C05348=1007.461,339.747,-160.298,169.990,53.598,160.501
C05349=1007.467,339.963,-160.328,169.997,53.593,160.501
C05350=1007.472,340.179,-160.358,170.005,53.589,160.502
C05351=1007.477,340.395,-160.388,170.011,53.585,160.502
C05352=1007.482,340.611,-160.418,170.018,53.580,160.503
C05353=1007.489,340.859,-160.453,170.026,53.576,160.503
C05354=1007.495,341.106,-160.487,170.035,53.571,160.504
C05355=1007.501,341.354,-160.521,170.043,53.566,160.504
C05356=1007.507,341.601,-160.557,170.051,53.561,160.505
C05357=1007.513,341.849,-160.591,170.059,53.556,160.505
C05358=1007.519,342.097,-160.625,170.068,53.552,160.506
C05359=1007.526,342.344,-160.660,170.077,53.547,160.507
C05360=1007.532,342.591,-160.694,170.085,53.542,160.507
C05361=1007.537,342.840,-160.729,170.093,53.538,160.508
C05362=1007.543,343.086,-160.764,170.101,53.533,160.509
C05363=1007.550,343.334,-160.799,170.110,53.528,160.509
C05364=1007.557,343.582,-160.834,170.118,53.523,160.510
C05365=1007.562,343.829,-160.868,170.126,53.519,160.511
C05366=1007.569,344.077,-160.903,170.134,53.514,160.511
C05367=1007.575,344.325,-160.938,170.143,53.509,160.512
C05368=1007.581,344.571,-160.973,170.151,53.504,160.512
C05369=1007.588,344.819,-161.007,170.159,53.500,160.513
C05370=1007.594,345.067,-161.043,170.168,53.495,160.514
C05371=1007.600,345.314,-161.078,170.176,53.491,160.515
C05372=1007.606,345.562,-161.112,170.185,53.486,160.515
C05373=1007.612,345.809,-161.148,170.194,53.481,160.516
C05374=1007.619,346.057,-161.183,170.202,53.476,160.516
C05375=1007.625,346.304,-161.219,170.210,53.472,160.517
C05376=1007.631,346.551,-161.253,170.219,53.467,160.518
C05377=1007.637,346.799,-161.289,170.227,53.463,160.519
C05378=1007.644,347.046,-161.324,170.236,53.459,160.519
C05379=1007.651,347.294,-161.359,170.244,53.454,160.520
C05380=1007.657,347.542,-161.394,170.252,53.449,160.521
C05381=1007.663,347.789,-161.429,170.261,53.444,160.521
C05382=1007.669,348.037,-161.465,170.270,53.440,160.522
C05383=1007.676,348.283,-161.501,170.279,53.436,160.523
C05384=1007.682,348.530,-161.536,170.287,53.431,160.524
C05385=1007.366,346.389,-161.589,170.194,53.514,160.524
C05386=1007.359,346.142,-161.554,170.186,53.518,160.523
C05387=1007.353,345.894,-161.518,170.177,53.523,160.523
C05388=1007.347,345.647,-161.484,170.168,53.527,160.522
C05389=1007.341,345.399,-161.449,170.160,53.532,160.521
C05390=1007.334,345.152,-161.413,170.151,53.537,160.520
C05391=1007.328,344.905,-161.379,170.143,53.542,160.520
C05392=1007.322,344.657,-161.344,170.135,53.546,160.519
C05393=1007.316,344.410,-161.308,170.127,53.551,160.519
C05394=1007.310,344.162,-161.274,170.118,53.555,160.518
C05395=1007.303,343.915,-161.239,170.110,53.560,160.517
C05396=1007.297,343.667,-161.205,170.102,53.564,160.516
C05397=1007.291,343.420,-161.169,170.093,53.569,160.516
C05398=1007.285,343.172,-161.135,170.085,53.574,160.515
C05399=1007.279,342.925,-161.101,170.077,53.578,160.515
C05400=1007.272,342.677,-161.066,170.069,53.583,160.514
C05401=1007.266,342.429,-161.031,170.059,53.588,160.513
C05402=1007.261,342.182,-160.997,170.051,53.593,160.513
C05403=1007.254,341.934,-160.962,170.043,53.598,160.512
C05404=1007.248,341.687,-160.928,170.034,53.602,160.511
C05405=1007.241,341.439,-160.893,170.026,53.607,160.511
C05406=1007.236,341.192,-160.858,170.018,53.612,160.510
C05407=1007.230,340.944,-160.823,170.010,53.617,160.510
C05408=1007.224,340.697,-160.789,170.001,53.621,160.509
C05409=1007.218,340.450,-160.755,169.993,53.626,160.508
C05410=1007.208,340.070,-160.703,169.982,53.634,160.508
C05411=1007.199,339.691,-160.650,169.969,53.641,160.507
C05412=1007.190,339.311,-160.597,169.956,53.649,160.506
C05413=1007.180,338.932,-160.544,169.944,53.656,160.505
C05414=1007.175,338.684,-160.511,169.935,53.661,160.504
C05415=1007.169,338.437,-160.477,169.927,53.666,160.504
C05416=1007.163,338.188,-160.442,169.919,53.671,160.503
C05417=1007.157,337.941,-160.408,169.911,53.676,160.502
C05418=1007.152,337.694,-160.374,169.903,53.681,160.502
C05419=1007.145,337.446,-160.340,169.896,53.685,160.501
C05420=1007.139,337.198,-160.305,169.888,53.690,160.501
C05421=1007.134,336.951,-160.272,169.880,53.695,160.500
C05422=1007.128,336.703,-160.238,169.871,53.700,160.500
C05423=1007.122,336.456,-160.204,169.863,53.705,160.499
C05424=1007.115,336.208,-160.171,169.855,53.710,160.499
C05425=1007.109,335.960,-160.137,169.847,53.715,160.498
C05426=1007.104,335.713,-160.104,169.840,53.720,160.498
C05427=1007.098,335.465,-160.069,169.831,53.725,160.497
C05428=1007.092,335.217,-160.036,169.823,53.730,160.497
C05429=1007.086,334.969,-160.002,169.815,53.735,160.496
C05430=1007.080,334.721,-159.968,169.807,53.740,160.496
C05431=1007.074,334.474,-159.934,169.799,53.745,160.495
C05432=1007.069,334.226,-159.901,169.791,53.750,160.494
C05433=1007.062,333.979,-159.868,169.784,53.755,160.494
C05434=1007.057,333.731,-159.834,169.776,53.760,160.494
C05435=1007.051,333.484,-159.800,169.768,53.765,160.493
C05436=1007.045,333.236,-159.767,169.760,53.770,160.493
C05437=1007.040,332.988,-159.733,169.752,53.776,160.492
C05438=1007.034,332.740,-159.700,169.744,53.781,160.492
C05439=1007.028,332.493,-159.666,169.736,53.786,160.491
C05440=1007.023,332.245,-159.633,169.728,53.791,160.491
C05441=1007.017,331.997,-159.599,169.721,53.796,160.490
C05442=1007.011,331.750,-159.566,169.713,53.801,160.490
C05443=1007.005,331.502,-159.533,169.705,53.806,160.489
C05444=1006.999,331.255,-159.499,169.698,53.812,160.489
C05445=1006.994,331.007,-159.466,169.689,53.817,160.488
C05446=1006.988,330.759,-159.433,169.682,53.822,160.488
C05447=1006.982,330.511,-159.400,169.675,53.827,160.488
C05448=1006.976,330.263,-159.367,169.667,53.832,160.487
C05449=1006.972,330.016,-159.334,169.659,53.837,160.487
C05450=1006.965,329.768,-159.301,169.651,53.842,160.486
C05451=1006.960,329.520,-159.267,169.643,53.848,160.486
C05452=1006.954,329.273,-159.234,169.635,53.853,160.485
C05453=1006.948,329.025,-159.201,169.629,53.858,160.485
C05454=1006.942,328.777,-159.168,169.620,53.863,160.484
C05455=1006.937,328.530,-159.136,169.613,53.869,160.484
C05456=1006.931,328.282,-159.103,169.605,53.874,160.483
C05457=1006.926,328.034,-159.070,169.597,53.879,160.483
C05458=1006.919,327.786,-159.037,169.589,53.885,160.483
C05459=1006.915,327.538,-159.005,169.582,53.890,160.482
C05460=1006.909,327.290,-158.971,169.575,53.895,160.482
C05461=1006.903,327.043,-158.939,169.567,53.900,160.481
C05462=1006.897,326.795,-158.905,169.559,53.906,160.481
C05463=1006.893,326.547,-158.873,169.552,53.911,160.481
C05464=1006.886,326.300,-158.840,169.544,53.916,160.480
C05465=1006.881,326.051,-158.808,169.537,53.922,160.480
C05466=1006.876,325.804,-158.775,169.529,53.927,160.480
C05467=1006.870,325.556,-158.742,169.521,53.932,160.479
C05468=1006.865,325.308,-158.710,169.514,53.938,160.479
C05469=1006.859,325.061,-158.677,169.507,53.943,160.478
C05470=1006.852,324.704,-158.630,169.495,53.951,160.478
C05471=1006.844,324.349,-158.583,169.485,53.959,160.477
C05472=1006.835,323.993,-158.538,169.474,53.967,160.477
C05473=1006.827,323.638,-158.491,169.464,53.974,160.476
C05474=1006.822,323.391,-158.460,169.456,53.980,160.476
C05475=1006.816,323.142,-158.428,169.449,53.985,160.476
C05476=1006.810,322.895,-158.396,169.441,53.990,160.475
C05477=1006.805,322.646,-158.363,169.434,53.996,160.475
C05478=1006.800,322.399,-158.332,169.426,54.001,160.474
C05479=1006.794,322.151,-158.300,169.419,54.007,160.474
C05480=1006.788,321.903,-158.268,169.411,54.013,160.474
C05481=1006.782,321.655,-158.236,169.404,54.018,160.474
C05482=1006.778,321.407,-158.204,169.397,54.024,160.473
C05483=1006.772,321.159,-158.172,169.389,54.029,160.473
C05484=1006.766,320.911,-158.140,169.382,54.035,160.473
C05485=1006.760,320.663,-158.108,169.375,54.040,160.472
C05486=1006.755,320.416,-158.076,169.367,54.046,160.472
C05487=1006.749,320.168,-158.045,169.360,54.051,160.472
C05488=1006.744,319.920,-158.012,169.353,54.057,160.471
C05489=1006.739,319.672,-157.980,169.345,54.062,160.471
C05490=1006.733,319.424,-157.949,169.338,54.068,160.471
C05491=1006.727,319.176,-157.917,169.330,54.074,160.470
C05492=1006.722,318.928,-157.886,169.324,54.079,160.470
C05493=1006.717,318.681,-157.854,169.316,54.085,160.470
C05494=1006.712,318.432,-157.821,169.308,54.090,160.469
C05495=1006.706,318.185,-157.790,169.302,54.096,160.469
C05496=1006.701,317.937,-157.758,169.294,54.101,160.469
C05497=1006.696,317.689,-157.727,169.287,54.108,160.469
C05498=1006.690,317.441,-157.695,169.280,54.113,160.468
C05499=1006.685,317.193,-157.663,169.273,54.118,160.468
C05500=1006.680,316.945,-157.632,169.265,54.124,160.468
C05501=1006.675,316.697,-157.600,169.258,54.129,160.467
C05502=1006.669,316.450,-157.569,169.251,54.135,160.467
C05503=1006.664,316.202,-157.538,169.244,54.141,160.467
C05504=1006.658,315.953,-157.506,169.237,54.147,160.467
C05505=1006.654,315.705,-157.474,169.229,54.152,160.466
C05506=1006.649,315.457,-157.442,169.223,54.158,160.466
C05507=1006.643,315.209,-157.411,169.215,54.163,160.466
C05508=1006.638,314.962,-157.380,169.208,54.170,160.466
C05509=1006.633,314.714,-157.348,169.201,54.175,160.465
C05510=1006.628,314.466,-157.317,169.194,54.181,160.465
C05511=1006.623,314.218,-157.286,169.187,54.187,160.465
C05512=1006.618,313.970,-157.254,169.180,54.192,160.465
C05513=1006.613,313.722,-157.223,169.172,54.198,160.464
C05514=1006.607,313.475,-157.191,169.166,54.204,160.464
C05515=1006.602,313.226,-157.160,169.159,54.210,160.464
C05516=1006.598,312.979,-157.128,169.152,54.215,160.464
C05517=1006.593,312.730,-157.097,169.145,54.221,160.464
C05518=1006.588,312.482,-157.066,169.137,54.227,160.463
C05519=1006.582,312.235,-157.035,169.130,54.232,160.463
C05520=1006.577,311.987,-157.004,169.123,54.238,160.463
C05521=1006.572,311.739,-156.973,169.117,54.244,160.463
C05522=1006.568,311.490,-156.941,169.110,54.250,160.462
C05523=1006.562,311.243,-156.910,169.102,54.256,160.462
C05524=1006.557,310.994,-156.879,169.095,54.261,160.462
C05525=1006.553,310.747,-156.848,169.088,54.267,160.462
C05526=1006.548,310.499,-156.817,169.082,54.273,160.461
C05527=1006.543,310.251,-156.786,169.074,54.279,160.461
C05528=1006.538,310.003,-156.754,169.068,54.284,160.461
C05529=1006.533,309.755,-156.723,169.061,54.291,160.461
C05530=1006.526,309.405,-156.679,169.051,54.299,160.461
C05531=1006.519,309.055,-156.635,169.041,54.307,160.460
C05532=1006.512,308.706,-156.592,169.032,54.316,160.460
C05533=1006.505,308.356,-156.549,169.022,54.324,160.460
C05534=1006.501,308.107,-156.517,169.015,54.329,160.460
C05535=1006.496,307.860,-156.487,169.008,54.336,160.459
C05536=1006.491,307.612,-156.456,169.000,54.341,160.459
C05537=1006.485,307.364,-156.426,168.994,54.347,160.459
C05538=1006.481,307.116,-156.396,168.987,54.354,160.459
C05539=1006.475,306.868,-156.366,168.981,54.359,160.459
C05540=1006.470,306.620,-156.335,168.973,54.365,160.458
C05541=1006.465,306.373,-156.306,168.967,54.371,160.458
C05542=1006.460,306.124,-156.275,168.960,54.377,160.458
C05543=1006.454,305.876,-156.245,168.954,54.383,160.458
C05544=1006.449,305.628,-156.214,168.946,54.389,160.458
C05545=1006.444,305.380,-156.185,168.939,54.396,160.458
C05546=1006.440,305.122,-156.153,168.933,54.401,160.458
C05547=1006.434,304.865,-156.122,168.926,54.407,160.457
C05548=1006.429,304.606,-156.090,168.918,54.414,160.457
C05549=1006.423,304.348,-156.059,168.911,54.420,160.457
C05550=1006.180,304.930,-156.495,168.907,54.441,160.461
C05551=1006.187,305.298,-156.541,168.917,54.432,160.461
C05552=1006.194,305.666,-156.585,168.927,54.424,160.461
C05553=1006.203,306.035,-156.630,168.937,54.414,160.462
C05554=1006.210,306.403,-156.675,168.948,54.405,160.462
C05555=1006.215,306.650,-156.705,168.954,54.399,160.462
C05556=1006.220,306.899,-156.735,168.962,54.394,160.462
C05557=1006.225,307.147,-156.765,168.968,54.388,160.462
C05558=1006.229,307.395,-156.795,168.975,54.381,160.463
C05559=1006.235,307.643,-156.825,168.982,54.376,160.463
C05560=1006.240,307.891,-156.856,168.989,54.370,160.463
C05561=1006.245,308.138,-156.887,168.995,54.364,160.463
C05562=1006.250,308.386,-156.918,169.003,54.358,160.463
C05563=1006.257,308.739,-156.961,169.012,54.350,160.464
C05564=1006.264,309.090,-157.005,169.022,54.342,160.464
C05565=1006.270,309.442,-157.050,169.032,54.334,160.464
C05566=1006.277,309.795,-157.093,169.042,54.326,160.465
C05567=1006.282,310.043,-157.124,169.049,54.319,160.465
C05568=1006.287,310.291,-157.155,169.056,54.314,160.465
C05569=1006.293,310.539,-157.187,169.063,54.308,160.466
C05570=1006.296,310.786,-157.218,169.069,54.302,160.465
C05571=1006.301,311.035,-157.249,169.077,54.297,160.466
C05572=1006.306,311.283,-157.280,169.083,54.291,160.466
C05573=1006.312,311.531,-157.311,169.091,54.285,160.466
C05574=1006.317,311.779,-157.342,169.097,54.280,160.467
C05575=1006.321,312.027,-157.374,169.104,54.273,160.467
C05576=1006.326,312.274,-157.404,169.111,54.268,160.467
C05577=1006.331,312.522,-157.435,169.119,54.262,160.467
C05578=1006.336,312.770,-157.467,169.125,54.256,160.467
C05579=1006.341,313.018,-157.498,169.133,54.251,160.468
C05580=1006.346,313.266,-157.529,169.140,54.245,160.468
C05581=1006.351,313.514,-157.561,169.147,54.240,160.468
C05582=1006.356,313.762,-157.592,169.154,54.233,160.468
C05583=1006.361,314.010,-157.623,169.161,54.228,160.469
C05584=1006.367,314.258,-157.655,169.168,54.222,160.469
C05585=1006.372,314.506,-157.686,169.175,54.217,160.469
C05586=1006.377,314.753,-157.717,169.182,54.211,160.469
C05587=1006.381,315.002,-157.749,169.190,54.205,160.470
C05588=1006.387,315.249,-157.781,169.196,54.200,160.470
C05589=1006.392,315.497,-157.812,169.204,54.194,160.470
C05590=1006.397,315.745,-157.843,169.210,54.189,160.471
C05591=1006.402,315.993,-157.874,169.218,54.183,160.471
C05592=1006.408,316.242,-157.907,169.225,54.177,160.471
C05593=1006.413,316.490,-157.938,169.232,54.172,160.471
C05594=1006.418,316.737,-157.969,169.239,54.166,160.472
C05595=1006.423,316.985,-158.000,169.247,54.160,160.472
C05596=1006.428,317.233,-158.032,169.254,54.155,160.472
C05597=1006.434,317.480,-158.064,169.261,54.149,160.473
C05598=1006.439,317.730,-158.096,169.268,54.144,160.473
C05599=1006.444,317.977,-158.127,169.276,54.138,160.473
C05600=1006.450,318.225,-158.159,169.283,54.133,160.474
C05601=1006.455,318.473,-158.190,169.290,54.127,160.474
C05602=1006.460,318.720,-158.221,169.298,54.122,160.474
C05603=1006.466,318.968,-158.253,169.305,54.116,160.475
C05604=1006.471,319.216,-158.286,169.312,54.111,160.475
C05605=1006.476,319.464,-158.317,169.319,54.105,160.475
C05606=1006.482,319.713,-158.349,169.327,54.099,160.476
C05607=1006.487,319.960,-158.380,169.334,54.094,160.476
C05608=1006.493,320.208,-158.412,169.341,54.088,160.476
C05609=1006.498,320.456,-158.445,169.349,54.083,160.477
C05610=1006.503,320.704,-158.476,169.356,54.078,160.477
C05611=1006.509,320.951,-158.508,169.363,54.072,160.477
C05612=1006.515,321.199,-158.540,169.371,54.066,160.478
C05613=1006.520,321.447,-158.572,169.378,54.061,160.478
C05614=1006.526,321.695,-158.604,169.385,54.055,160.478
C05615=1006.531,321.943,-158.636,169.393,54.050,160.478
C05616=1006.536,322.190,-158.668,169.401,54.045,160.479
C05617=1006.542,322.439,-158.700,169.407,54.039,160.479
C05618=1006.547,322.686,-158.731,169.415,54.034,160.480
C05619=1006.553,322.934,-158.763,169.423,54.028,160.480
C05620=1006.558,323.182,-158.796,169.430,54.022,160.480
C05621=1006.564,323.430,-158.828,169.437,54.017,160.481
C05622=1006.569,323.678,-158.859,169.445,54.012,160.481
C05623=1006.578,324.036,-158.905,169.456,54.004,160.482
C05624=1006.586,324.394,-158.952,169.466,53.997,160.482
C05625=1006.594,324.752,-158.998,169.478,53.989,160.483
C05626=1006.602,325.110,-159.046,169.489,53.981,160.483
C05627=1006.607,325.358,-159.078,169.495,53.976,160.484
C05628=1006.613,325.605,-159.111,169.503,53.971,160.484
C05629=1006.618,325.854,-159.143,169.511,53.965,160.485
C05630=1006.623,326.101,-159.176,169.519,53.959,160.485
C05631=1006.629,326.348,-159.209,169.526,53.955,160.485
C05632=1006.635,326.597,-159.242,169.533,53.949,160.486
C05633=1006.639,326.844,-159.275,169.542,53.944,160.486
C05634=1006.645,327.092,-159.307,169.549,53.938,160.487
C05635=1006.651,327.340,-159.340,169.556,53.933,160.487
C05636=1006.657,327.587,-159.372,169.564,53.928,160.487
C05637=1006.662,327.836,-159.405,169.572,53.923,160.488
C05638=1006.668,328.084,-159.438,169.580,53.918,160.488
C05639=1006.674,328.331,-159.471,169.587,53.912,160.489
C05640=1006.679,328.578,-159.504,169.594,53.907,160.489
C05641=1006.684,328.827,-159.537,169.602,53.902,160.489
C05642=1006.690,329.075,-159.570,169.610,53.897,160.490
C05643=1006.696,329.322,-159.603,169.618,53.891,160.490
C05644=1006.701,329.570,-159.636,169.626,53.886,160.491
C05645=1006.707,329.817,-159.669,169.633,53.882,160.491
C05646=1006.713,330.065,-159.702,169.641,53.876,160.492
C05647=1006.719,330.313,-159.735,169.649,53.871,160.492
C05648=1006.725,330.561,-159.768,169.656,53.865,160.493
C05649=1006.730,330.809,-159.801,169.664,53.860,160.493
C05650=1006.736,331.056,-159.834,169.672,53.856,160.494
C05651=1006.741,331.303,-159.867,169.679,53.850,160.494
C05652=1006.747,331.551,-159.900,169.687,53.845,160.495
C05653=1006.752,331.799,-159.934,169.695,53.840,160.495
C05654=1006.758,332.047,-159.967,169.703,53.835,160.496
C05655=1006.764,332.295,-160.000,169.711,53.830,160.496
C05656=1006.769,332.542,-160.034,169.718,53.825,160.497
C05657=1006.775,332.790,-160.068,169.726,53.820,160.497
C05658=1006.780,333.038,-160.101,169.734,53.815,160.498
C05659=1006.787,333.286,-160.134,169.742,53.809,160.498
C05660=1006.793,333.533,-160.168,169.750,53.804,160.499
C05661=1006.798,333.781,-160.201,169.758,53.800,160.499
C05662=1006.804,334.029,-160.235,169.766,53.795,160.500
C05663=1006.810,334.276,-160.269,169.774,53.790,160.500
C05664=1006.815,334.524,-160.302,169.782,53.785,160.501
C05665=1006.821,334.771,-160.336,169.789,53.779,160.501
C05666=1006.827,335.019,-160.369,169.797,53.774,160.502
C05667=1006.833,335.268,-160.403,169.805,53.769,160.502
C05668=1006.839,335.515,-160.437,169.813,53.765,160.503
C05669=1006.845,335.763,-160.470,169.822,53.760,160.503
C05670=1006.851,336.010,-160.504,169.830,53.755,160.504
C05671=1006.857,336.257,-160.538,169.838,53.750,160.504
C05672=1006.862,336.505,-160.571,169.846,53.745,160.505
C05673=1006.869,336.753,-160.606,169.854,53.740,160.506
C05674=1006.874,337.001,-160.639,169.862,53.735,160.506
C05675=1006.880,337.248,-160.673,169.870,53.730,160.507
C05676=1006.886,337.496,-160.707,169.877,53.725,160.507
C05677=1006.892,337.744,-160.742,169.885,53.720,160.508
C05678=1006.898,337.991,-160.775,169.893,53.715,160.508
C05679=1006.904,338.239,-160.809,169.902,53.710,160.509
C05680=1006.910,338.486,-160.843,169.910,53.706,160.510
C05681=1006.916,338.734,-160.877,169.918,53.701,160.510
C05682=1006.921,338.982,-160.912,169.926,53.696,160.511
C05683=1006.929,339.306,-160.957,169.937,53.689,160.511
C05684=1006.937,339.630,-161.001,169.948,53.683,160.512
C05685=1006.945,339.955,-161.047,169.958,53.677,160.513
C05686=1006.953,340.279,-161.091,169.969,53.671,160.514
C05687=1006.959,340.527,-161.126,169.977,53.666,160.515
C05688=1006.964,340.774,-161.161,169.985,53.661,160.515
C05689=1006.971,341.022,-161.195,169.994,53.656,160.516
C05690=1006.977,341.270,-161.229,170.002,53.651,160.516
C05691=1006.983,341.518,-161.263,170.010,53.647,160.517
C05692=1006.989,341.765,-161.297,170.018,53.642,160.518
C05693=1006.995,342.013,-161.333,170.026,53.637,160.518
C05694=1007.001,342.260,-161.367,170.035,53.633,160.519
C05695=1007.007,342.508,-161.402,170.043,53.628,160.519
C05696=1007.013,342.755,-161.436,170.052,53.624,160.520
C05697=1007.020,343.003,-161.471,170.060,53.619,160.521
C05698=1007.025,343.250,-161.506,170.068,53.614,160.521
C05699=1007.032,343.498,-161.541,170.076,53.610,160.522
C05700=1007.038,343.745,-161.575,170.085,53.605,160.523
C05701=1007.044,343.993,-161.609,170.093,53.600,160.523
C05702=1007.050,344.240,-161.645,170.102,53.595,160.524
C05703=1006.736,342.085,-161.703,170.011,53.676,160.524
C05704=1006.730,341.839,-161.668,170.002,53.680,160.523
C05705=1006.724,341.591,-161.634,169.994,53.685,160.523
C05706=1006.718,341.343,-161.599,169.986,53.690,160.522
C05707=1006.713,341.096,-161.565,169.978,53.695,160.521
C05708=1006.706,340.848,-161.530,169.970,53.700,160.521
C05709=1006.700,340.600,-161.496,169.961,53.704,160.520
C05710=1006.694,340.353,-161.462,169.953,53.709,160.520
C05711=1006.688,340.105,-161.428,169.945,53.714,160.519
C05712=1006.682,339.837,-161.391,169.936,53.719,160.518
C05713=1006.676,339.568,-161.353,169.927,53.725,160.518
C05714=1006.669,339.300,-161.315,169.918,53.729,160.517
C05715=1006.663,339.031,-161.279,169.909,53.734,160.516
C05716=1006.657,338.784,-161.245,169.901,53.739,160.516
C05717=1006.651,338.536,-161.211,169.893,53.744,160.515
C05718=1006.645,338.289,-161.177,169.885,53.749,160.515
C05719=1006.639,338.041,-161.143,169.876,53.754,160.514
C05720=1006.633,337.794,-161.109,169.868,53.758,160.513
C05721=1006.628,337.545,-161.074,169.860,53.763,160.513
C05722=1006.622,337.298,-161.040,169.853,53.768,160.512
C05723=1006.616,337.050,-161.006,169.845,53.773,160.512
C05724=1006.610,336.803,-160.973,169.837,53.778,160.511
C05725=1006.604,336.556,-160.939,169.828,53.783,160.510
C05726=1006.597,336.307,-160.906,169.820,53.788,160.510
C05727=1006.592,336.060,-160.872,169.812,53.793,160.509
C05728=1006.586,335.812,-160.838,169.804,53.798,160.509
C05729=1006.580,335.565,-160.804,169.796,53.803,160.508
C05730=1006.575,335.317,-160.771,169.788,53.808,160.508
C05731=1006.569,335.069,-160.737,169.780,53.813,160.507
C05732=1006.563,334.821,-160.703,169.773,53.817,160.507
C05733=1006.557,334.574,-160.669,169.765,53.822,160.506
C05734=1006.551,334.327,-160.637,169.757,53.827,160.505
C05735=1006.546,334.079,-160.603,169.748,53.832,160.505
C05736=1006.540,333.831,-160.569,169.740,53.837,160.504
C05737=1006.534,333.583,-160.536,169.733,53.843,160.504
C05738=1006.529,333.336,-160.503,169.725,53.848,160.503
C05739=1006.523,333.088,-160.469,169.716,53.853,160.503
C05740=1006.517,332.840,-160.435,169.709,53.857,160.502
C05741=1006.512,332.592,-160.402,169.701,53.862,160.502
C05742=1006.506,332.345,-160.369,169.693,53.867,160.501
C05743=1006.500,332.097,-160.335,169.686,53.873,160.501
C05744=1006.494,331.849,-160.302,169.677,53.878,160.500
C05745=1006.489,331.601,-160.269,169.670,53.882,160.500
C05746=1006.483,331.354,-160.235,169.662,53.887,160.499
C05747=1006.477,331.106,-160.202,169.654,53.892,160.499
C05748=1006.472,330.858,-160.168,169.646,53.898,160.498
C05749=1006.467,330.611,-160.135,169.638,53.903,160.498
C05750=1006.460,330.363,-160.103,169.630,53.908,160.497
C05751=1006.455,330.115,-160.070,169.624,53.913,160.497
C05752=1006.449,329.867,-160.037,169.616,53.918,160.496
C05753=1006.443,329.619,-160.004,169.607,53.923,160.496
C05754=1006.438,329.372,-159.971,169.600,53.929,160.495
C05755=1006.432,329.124,-159.938,169.592,53.934,160.495
C05756=1006.427,328.876,-159.906,169.585,53.939,160.495
C05757=1006.421,328.628,-159.872,169.577,53.944,160.494
C05758=1006.416,328.381,-159.840,169.569,53.949,160.493
C05759=1006.410,328.133,-159.807,169.561,53.954,160.493
C05760=1006.405,327.885,-159.774,169.554,53.959,160.493
C05761=1006.399,327.638,-159.742,169.547,53.965,160.492
C05762=1006.394,327.390,-159.708,169.538,53.970,160.492
C05763=1006.388,327.142,-159.676,169.531,53.975,160.491
C05764=1006.383,326.894,-159.643,169.524,53.980,160.491
C05765=1006.377,326.646,-159.611,169.516,53.986,160.491
C05766=1006.371,326.398,-159.578,169.508,53.991,160.490
C05767=1006.366,326.151,-159.546,169.500,53.996,160.490
C05768=1006.361,325.903,-159.512,169.493,54.001,160.489
C05769=1006.355,325.656,-159.480,169.486,54.006,160.489
C05770=1006.350,325.407,-159.447,169.478,54.012,160.488
C05771=1006.345,325.159,-159.415,169.470,54.017,160.488
C05772=1006.337,324.799,-159.367,169.460,54.025,160.487
C05773=1006.329,324.439,-159.320,169.448,54.033,160.487
C05774=1006.321,324.078,-159.274,169.437,54.041,160.486
C05775=1006.312,323.719,-159.228,169.427,54.048,160.486
C05776=1006.307,323.470,-159.195,169.419,54.053,160.485
C05777=1006.302,323.222,-159.163,169.411,54.059,160.485
C05778=1006.296,322.974,-159.131,169.405,54.064,160.485
C05779=1006.290,322.727,-159.100,169.397,54.070,160.484
C05780=1006.284,322.479,-159.068,169.389,54.075,160.484
C05781=1006.280,322.231,-159.035,169.381,54.080,160.483
C05782=1006.274,321.983,-159.004,169.375,54.086,160.483
C05783=1006.268,321.735,-158.972,169.367,54.091,160.483
C05784=1006.263,321.487,-158.940,169.360,54.097,160.482
C05785=1006.257,321.239,-158.908,169.352,54.102,160.482
C05786=1006.252,320.992,-158.876,169.345,54.107,160.481
C05787=1006.247,320.744,-158.844,169.337,54.113,160.481
C05788=1006.241,320.496,-158.812,169.331,54.118,160.481
C05789=1006.235,320.248,-158.780,169.323,54.124,160.480
C05790=1006.230,320.000,-158.750,169.315,54.129,160.480
C05791=1006.224,319.752,-158.718,169.309,54.135,160.480
C05792=1006.219,319.504,-158.686,169.301,54.140,160.479
C05793=1006.214,319.257,-158.654,169.293,54.145,160.479
C05794=1006.209,319.009,-158.622,169.286,54.151,160.479
C05795=1006.203,318.760,-158.591,169.279,54.156,160.478
C05796=1006.198,318.513,-158.559,169.271,54.162,160.478
C05797=1006.193,318.265,-158.527,169.264,54.167,160.478
C05798=1006.188,318.017,-158.496,169.257,54.173,160.477
C05799=1006.183,317.769,-158.464,169.250,54.178,160.477
C05800=1006.177,317.521,-158.432,169.242,54.184,160.477
C05801=1006.172,317.273,-158.401,169.235,54.190,160.476
C05802=1006.166,317.025,-158.369,169.228,54.195,160.476
C05803=1006.161,316.777,-158.339,169.221,54.201,160.476
C05804=1006.157,316.529,-158.306,169.214,54.206,160.475
C05805=1006.152,316.281,-158.275,169.206,54.212,160.475
C05806=1006.146,316.034,-158.244,169.199,54.218,160.475
C05807=1006.141,315.786,-158.213,169.193,54.223,160.475
C05808=1006.136,315.538,-158.181,169.185,54.229,160.474
C05809=1006.131,315.290,-158.150,169.178,54.234,160.474
C05810=1006.126,315.042,-158.118,169.171,54.240,160.474
C05811=1006.121,314.794,-158.087,169.163,54.246,160.473
C05812=1006.116,314.546,-158.055,169.156,54.251,160.473
C05813=1006.110,314.298,-158.024,169.149,54.257,160.473
C05814=1006.105,314.050,-157.993,169.143,54.262,160.473
C05815=1006.101,313.802,-157.961,169.135,54.268,160.472
C05816=1006.096,313.554,-157.930,169.128,54.273,160.472
C05817=1006.091,313.306,-157.899,169.121,54.279,160.472
C05818=1006.085,313.059,-157.868,169.114,54.284,160.471
C05819=1006.080,312.810,-157.837,169.107,54.290,160.471
C05820=1006.075,312.562,-157.806,169.100,54.296,160.471
C05821=1006.071,312.314,-157.774,169.093,54.302,160.471
C05822=1006.065,312.066,-157.742,169.086,54.307,160.470
C05823=1006.061,311.819,-157.712,169.079,54.313,160.470
C05824=1006.056,311.571,-157.681,169.071,54.319,160.470
C05825=1006.051,311.323,-157.650,169.065,54.324,160.470
C05826=1006.046,311.074,-157.618,169.057,54.330,160.469
C05827=1006.041,310.826,-157.587,169.051,54.336,160.469
C05828=1006.036,310.578,-157.557,169.043,54.342,160.469
C05829=1006.031,310.331,-157.525,169.037,54.347,160.469
C05830=1006.026,310.083,-157.494,169.030,54.353,160.468
C05831=1006.021,309.835,-157.463,169.023,54.359,160.468
C05832=1006.015,309.480,-157.419,169.013,54.367,160.468
C05833=1006.008,309.126,-157.375,169.004,54.375,160.468
C05834=1006.002,308.772,-157.331,168.993,54.383,160.467
C05835=1005.994,308.417,-157.287,168.984,54.391,160.467
C05836=1005.989,308.169,-157.256,168.977,54.398,160.467
C05837=1005.985,307.922,-157.225,168.970,54.403,160.466
C05838=1005.980,307.673,-157.194,168.963,54.409,160.466
C05839=1005.975,307.426,-157.165,168.956,54.415,160.466
C05840=1005.970,307.184,-157.135,168.949,54.421,160.466
C05841=1005.965,306.942,-157.105,168.942,54.426,160.466
C05842=1005.960,306.700,-157.076,168.936,54.432,160.465
C05843=1005.955,306.459,-157.047,168.930,54.438,160.465
C05844=1005.950,306.217,-157.017,168.922,54.443,160.465
C05845=1005.945,305.976,-156.988,168.916,54.449,160.465
C05846=1005.941,305.734,-156.959,168.909,54.455,160.465
C05847=1005.935,305.492,-156.930,168.902,54.461,160.464
C05848=1005.691,306.038,-157.362,168.898,54.480,160.468
C05849=1005.698,306.392,-157.405,168.908,54.471,160.468
C05850=1005.705,306.747,-157.447,168.918,54.463,160.468
C05851=1005.713,307.102,-157.491,168.928,54.454,160.469
C05852=1005.719,307.456,-157.534,168.937,54.446,160.469
C05853=1005.725,307.704,-157.564,168.944,54.441,160.469
C05854=1005.730,307.952,-157.595,168.951,54.434,160.469
C05855=1005.735,308.200,-157.626,168.958,54.429,160.470
C05856=1005.739,308.448,-157.656,168.965,54.423,160.470
C05857=1005.746,308.805,-157.700,168.975,54.415,160.470
C05858=1005.753,309.162,-157.744,168.985,54.407,160.471
C05859=1005.760,309.517,-157.789,168.994,54.398,160.471
C05860=1005.766,309.874,-157.834,169.004,54.390,160.471
C05861=1005.772,310.122,-157.865,169.012,54.384,160.472
C05862=1005.777,310.370,-157.896,169.018,54.379,160.472
C05863=1005.781,310.619,-157.927,169.026,54.373,160.472
C05864=1005.785,310.866,-157.958,169.032,54.367,160.472
C05865=1005.790,311.114,-157.989,169.040,54.362,160.473
C05866=1005.796,311.362,-158.020,169.046,54.356,160.473
C05867=1005.801,311.611,-158.051,169.053,54.351,160.473
C05868=1005.805,311.859,-158.082,169.061,54.345,160.474
C05869=1005.809,312.106,-158.113,169.067,54.339,160.474
C05870=1005.815,312.354,-158.144,169.074,54.334,160.474
C05871=1005.820,312.602,-158.175,169.081,54.328,160.474
C05872=1005.825,312.850,-158.206,169.089,54.323,160.475
C05873=1005.830,313.098,-158.237,169.095,54.317,160.475
C05874=1005.834,313.347,-158.269,169.103,54.312,160.475
C05875=1005.839,313.594,-158.300,169.109,54.306,160.475
C05876=1005.844,313.842,-158.331,169.117,54.300,160.476
C05877=1005.849,314.090,-158.362,169.124,54.294,160.476
C05878=1005.855,314.337,-158.394,169.131,54.289,160.476
C05879=1005.860,314.586,-158.425,169.139,54.283,160.477
C05880=1005.864,314.834,-158.456,169.145,54.278,160.477
C05881=1005.870,315.081,-158.488,169.153,54.272,160.477
C05882=1005.875,315.330,-158.519,169.160,54.267,160.478
C05883=1005.880,315.578,-158.550,169.167,54.262,160.478
C05884=1005.885,315.825,-158.581,169.174,54.256,160.478
C05885=1005.889,316.074,-158.613,169.181,54.251,160.479
C05886=1005.895,316.321,-158.644,169.188,54.245,160.479
C05887=1005.900,316.569,-158.675,169.196,54.240,160.479
C05888=1005.905,316.817,-158.707,169.203,54.234,160.480
C05889=1005.911,317.066,-158.738,169.210,54.229,160.480
C05890=1005.916,317.313,-158.770,169.218,54.223,160.480
C05891=1005.921,317.562,-158.802,169.224,54.218,160.480
C05892=1005.926,317.809,-158.833,169.232,54.212,160.481
C05893=1005.931,318.057,-158.865,169.239,54.206,160.481
C05894=1005.937,318.305,-158.896,169.246,54.201,160.481
C05895=1005.942,318.552,-158.928,169.254,54.195,160.482
C05896=1005.947,318.801,-158.960,169.260,54.190,160.482
C05897=1005.952,319.049,-158.991,169.268,54.184,160.482
C05898=1005.958,319.296,-159.023,169.276,54.179,160.483
C05899=1005.963,319.544,-159.054,169.283,54.174,160.483
C05900=1005.969,319.793,-159.086,169.290,54.168,160.484
C05901=1005.974,320.040,-159.117,169.297,54.163,160.484
C05902=1005.979,320.288,-159.150,169.305,54.157,160.484
C05903=1005.984,320.536,-159.181,169.312,54.152,160.485
C05904=1005.990,320.785,-159.213,169.319,54.147,160.485
C05905=1005.995,321.032,-159.244,169.327,54.141,160.485
C05906=1006.001,321.280,-159.276,169.335,54.136,160.486
C05907=1006.006,321.528,-159.309,169.341,54.131,160.486
C05908=1006.011,321.776,-159.340,169.349,54.126,160.487
C05909=1006.017,322.023,-159.372,169.357,54.120,160.487
C05910=1006.023,322.271,-159.404,169.364,54.115,160.487
C05911=1006.028,322.519,-159.436,169.371,54.109,160.488
C05912=1006.034,322.767,-159.468,169.379,54.104,160.488
C05913=1006.039,323.015,-159.500,169.386,54.099,160.489
C05914=1006.044,323.262,-159.532,169.394,54.093,160.489
C05915=1006.050,323.511,-159.564,169.402,54.088,160.489
C05916=1006.055,323.758,-159.595,169.409,54.082,160.490
C05917=1006.064,324.121,-159.641,169.419,54.075,160.490
C05918=1006.072,324.484,-159.689,169.431,54.067,160.491
C05919=1006.080,324.846,-159.737,169.442,54.059,160.492
C05920=1006.087,325.209,-159.784,169.452,54.052,160.492
C05921=1006.093,325.457,-159.816,169.460,54.046,160.493
C05922=1006.098,325.705,-159.849,169.468,54.041,160.493
C05923=1006.104,325.953,-159.882,169.476,54.036,160.494
C05924=1006.109,326.200,-159.914,169.483,54.031,160.494
C05925=1006.114,326.448,-159.947,169.491,54.025,160.494
C05926=1006.119,326.696,-159.979,169.499,54.020,160.495
C05927=1006.125,326.943,-160.012,169.505,54.015,160.495
C05928=1006.131,327.192,-160.045,169.513,54.010,160.496
C05929=1006.136,327.439,-160.077,169.521,54.005,160.496
C05930=1006.142,327.687,-160.110,169.529,54.000,160.497
C05931=1006.147,327.935,-160.143,169.536,53.995,160.497
C05932=1006.153,328.182,-160.175,169.544,53.989,160.498
C05933=1006.158,328.431,-160.208,169.552,53.984,160.498
C05934=1006.164,328.679,-160.241,169.560,53.979,160.498
C05935=1006.169,328.925,-160.274,169.567,53.974,160.499
C05936=1006.175,329.173,-160.307,169.575,53.969,160.500
C05937=1006.180,329.422,-160.340,169.582,53.963,160.500
C05938=1006.186,329.670,-160.372,169.591,53.958,160.500
C05939=1006.191,329.917,-160.405,169.598,53.954,160.501
C05940=1006.198,330.164,-160.438,169.606,53.949,160.502
C05941=1006.203,330.412,-160.472,169.613,53.943,160.502
C05942=1006.208,330.661,-160.504,169.622,53.938,160.502
C05943=1006.214,330.908,-160.537,169.630,53.933,160.503
C05944=1006.220,331.156,-160.570,169.637,53.929,160.504
C05945=1006.225,331.403,-160.603,169.644,53.923,160.504
C05946=1006.231,331.651,-160.637,169.652,53.918,160.504
C05947=1006.237,331.899,-160.671,169.661,53.913,160.505
C05948=1006.242,332.147,-160.704,169.669,53.908,160.506
C05949=1006.248,332.394,-160.737,169.676,53.904,160.506
C05950=1006.253,332.642,-160.770,169.684,53.899,160.507
C05951=1006.258,332.890,-160.804,169.691,53.893,160.507
C05952=1006.265,333.137,-160.836,169.700,53.888,160.508
C05953=1006.270,333.385,-160.870,169.708,53.883,160.508
C05954=1006.276,333.632,-160.904,169.715,53.878,160.509
C05955=1006.282,333.880,-160.937,169.723,53.873,160.509
C05956=1006.287,334.128,-160.970,169.731,53.868,160.510
C05957=1006.293,334.375,-161.004,169.739,53.863,160.510
C05958=1006.299,334.623,-161.038,169.747,53.858,160.511
C05959=1006.304,334.871,-161.071,169.755,53.854,160.512
C05960=1006.310,335.119,-161.105,169.763,53.849,160.512
C05961=1006.316,335.366,-161.138,169.771,53.844,160.513
C05962=1006.322,335.614,-161.171,169.779,53.839,160.513
C05963=1006.328,335.862,-161.206,169.787,53.834,160.514
C05964=1006.334,336.110,-161.239,169.795,53.829,160.514
C05965=1006.340,336.357,-161.273,169.803,53.824,160.515
C05966=1006.345,336.605,-161.306,169.811,53.819,160.515
C05967=1006.351,336.852,-161.340,169.819,53.814,160.516
C05968=1006.357,337.100,-161.374,169.828,53.810,160.517
C05969=1006.362,337.348,-161.408,169.836,53.805,160.517
C05970=1006.369,337.596,-161.442,169.844,53.800,160.518
C05971=1006.375,337.843,-161.476,169.851,53.795,160.518
C05972=1006.380,338.091,-161.510,169.859,53.790,160.519
C05973=1006.386,338.338,-161.544,169.867,53.785,160.520
C05974=1006.392,338.585,-161.578,169.876,53.781,160.520
C05975=1006.398,338.834,-161.611,169.884,53.776,160.521
C05976=1006.403,339.082,-161.646,169.892,53.771,160.521
C05977=1006.409,339.293,-161.675,169.900,53.767,160.522
C05978=1006.413,339.505,-161.704,169.906,53.763,160.522
C05979=1006.419,339.717,-161.734,169.913,53.759,160.523
C05980=1006.424,339.930,-161.763,169.920,53.755,160.524
C05981=1006.113,337.770,-161.827,169.831,53.833,160.523
C05982=1006.107,337.523,-161.793,169.823,53.838,160.522
C05983=1006.102,337.275,-161.758,169.814,53.842,160.522
C05984=1006.096,337.027,-161.725,169.806,53.847,160.521
C05985=1006.090,336.779,-161.690,169.799,53.852,160.521
C05986=1006.084,336.532,-161.658,169.791,53.857,160.520
C05987=1006.078,336.284,-161.624,169.783,53.862,160.519
C05988=1006.072,336.036,-161.590,169.774,53.867,160.519
C05989=1006.067,335.789,-161.557,169.766,53.872,160.518
C05990=1006.061,335.541,-161.523,169.758,53.876,160.517
C05991=1006.056,335.293,-161.490,169.750,53.881,160.517
C05992=1006.050,335.046,-161.456,169.742,53.886,160.516
C05993=1006.044,334.798,-161.422,169.734,53.890,160.516
C05994=1006.039,334.550,-161.389,169.726,53.895,160.515
C05995=1006.032,334.303,-161.356,169.718,53.900,160.515
C05996=1006.026,334.055,-161.322,169.710,53.905,160.514
C05997=1006.021,333.808,-161.289,169.702,53.910,160.513
C05998=1006.015,333.560,-161.255,169.694,53.915,160.513
C05999=1006.010,333.312,-161.222,169.687,53.920,160.512
C06000=1006.004,333.064,-161.189,169.679,53.925,160.512
C06001=1005.998,332.817,-161.155,169.671,53.930,160.511
C06002=1005.993,332.569,-161.121,169.662,53.935,160.511
C06003=1005.987,332.321,-161.088,169.654,53.940,160.510
C06004=1005.981,332.074,-161.056,169.648,53.945,160.510
C06005=1005.976,331.826,-161.022,169.640,53.950,160.509
C06006=1005.970,331.578,-160.989,169.632,53.955,160.509
C06007=1005.965,331.330,-160.956,169.623,53.960,160.508
C06008=1005.959,331.082,-160.922,169.616,53.965,160.508
C06009=1005.954,330.834,-160.889,169.608,53.970,160.507
C06010=1005.949,330.587,-160.856,169.600,53.975,160.506
C06011=1005.942,330.339,-160.823,169.592,53.980,160.506
C06012=1005.937,330.091,-160.791,169.584,53.985,160.506
C06013=1005.932,329.844,-160.758,169.577,53.990,160.505
C06014=1005.926,329.596,-160.725,169.569,53.995,160.504
C06015=1005.920,329.348,-160.692,169.562,54.001,160.504
C06016=1005.914,329.100,-160.660,169.553,54.006,160.504
C06017=1005.909,328.853,-160.627,169.546,54.010,160.503
C06018=1005.904,328.605,-160.593,169.538,54.015,160.502
C06019=1005.898,328.357,-160.561,169.531,54.021,160.502
C06020=1005.893,328.110,-160.528,169.523,54.025,160.502
C06021=1005.887,327.862,-160.495,169.515,54.030,160.501
C06022=1005.881,327.613,-160.463,169.508,54.036,160.501
C06023=1005.877,327.366,-160.430,169.500,54.041,160.500
C06024=1005.871,327.118,-160.398,169.493,54.046,160.500
C06025=1005.866,326.871,-160.365,169.485,54.051,160.499
C06026=1005.860,326.622,-160.332,169.477,54.056,160.499
C06027=1005.854,326.375,-160.300,169.470,54.061,160.498
C06028=1005.849,326.127,-160.267,169.462,54.066,160.498
C06029=1005.844,325.879,-160.234,169.454,54.072,160.497
C06030=1005.838,325.631,-160.202,169.447,54.077,160.497
C06031=1005.833,325.383,-160.170,169.439,54.082,160.496
C06032=1005.828,325.136,-160.137,169.432,54.087,160.496
C06033=1005.822,324.887,-160.105,169.423,54.092,160.495
C06034=1005.817,324.616,-160.069,169.416,54.098,160.495
C06035=1005.811,324.343,-160.033,169.407,54.104,160.495
C06036=1005.804,324.071,-159.998,169.400,54.110,160.494
C06037=1005.798,323.799,-159.964,169.391,54.116,160.494
C06038=1005.794,323.551,-159.931,169.384,54.120,160.493
C06039=1005.788,323.303,-159.899,169.376,54.126,160.493
C06040=1005.782,323.055,-159.868,169.368,54.131,160.492
C06041=1005.776,322.807,-159.836,169.361,54.136,160.492
C06042=1005.771,322.559,-159.804,169.354,54.142,160.492
C06043=1005.766,322.312,-159.772,169.346,54.147,160.491
C06044=1005.760,322.063,-159.740,169.339,54.152,160.491
C06045=1005.755,321.816,-159.708,169.331,54.158,160.490
C06046=1005.750,321.568,-159.677,169.323,54.163,160.490
C06047=1005.744,321.319,-159.645,169.317,54.168,160.490
C06048=1005.738,321.072,-159.613,169.309,54.174,160.489
C06049=1005.734,320.824,-159.581,169.302,54.179,160.489
C06050=1005.728,320.576,-159.549,169.294,54.184,160.488
C06051=1005.723,320.328,-159.518,169.287,54.190,160.488
C06052=1005.717,320.080,-159.487,169.280,54.195,160.488
C06053=1005.712,319.833,-159.455,169.272,54.200,160.487
C06054=1005.706,319.585,-159.423,169.264,54.206,160.487
C06055=1005.702,319.336,-159.391,169.258,54.211,160.486
C06056=1005.696,319.089,-159.360,169.250,54.217,160.486
C06057=1005.691,318.841,-159.328,169.243,54.222,160.486
C06058=1005.686,318.593,-159.297,169.235,54.227,160.485
C06059=1005.680,318.345,-159.265,169.229,54.232,160.485
C06060=1005.675,318.096,-159.233,169.221,54.238,160.485
C06061=1005.670,317.849,-159.202,169.213,54.244,160.484
C06062=1005.665,317.601,-159.171,169.207,54.249,160.484
C06063=1005.660,317.353,-159.139,169.199,54.255,160.484
C06064=1005.655,317.105,-159.108,169.193,54.260,160.483
C06065=1005.649,316.858,-159.077,169.185,54.266,160.483
C06066=1005.645,316.609,-159.045,169.178,54.270,160.482
C06067=1005.639,316.362,-159.013,169.170,54.276,160.482
C06068=1005.634,316.113,-158.982,169.164,54.281,160.482
C06069=1005.629,315.866,-158.951,169.156,54.287,160.481
C06070=1005.624,315.618,-158.920,169.148,54.293,160.481
C06071=1005.620,315.369,-158.888,169.142,54.298,160.481
C06072=1005.614,315.122,-158.857,169.134,54.304,160.480
C06073=1005.609,314.874,-158.826,169.127,54.309,160.480
C06074=1005.604,314.626,-158.795,169.120,54.315,160.480
C06075=1005.599,314.378,-158.763,169.113,54.320,160.479
C06076=1005.594,314.130,-158.732,169.106,54.326,160.479
C06077=1005.589,313.881,-158.701,169.099,54.331,160.479
C06078=1005.584,313.634,-158.669,169.091,54.337,160.478
C06079=1005.579,313.387,-158.638,169.085,54.342,160.478
C06080=1005.574,313.138,-158.607,169.077,54.348,160.478
C06081=1005.569,312.890,-158.576,169.070,54.353,160.478
C06082=1005.565,312.642,-158.545,169.063,54.359,160.477
C06083=1005.560,312.394,-158.514,169.057,54.365,160.477
C06084=1005.554,312.146,-158.482,169.050,54.370,160.477
C06085=1005.550,311.899,-158.452,169.042,54.376,160.476
C06086=1005.545,311.651,-158.421,169.036,54.381,160.476
C06087=1005.540,311.402,-158.390,169.028,54.387,160.476
C06088=1005.535,311.154,-158.358,169.022,54.392,160.476
C06089=1005.531,310.907,-158.328,169.014,54.398,160.475
C06090=1005.526,310.658,-158.297,169.008,54.404,160.475
C06091=1005.521,310.410,-158.266,169.000,54.409,160.475
C06092=1005.516,310.162,-158.235,168.993,54.415,160.474
C06093=1005.512,309.914,-158.204,168.986,54.420,160.474
C06094=1005.504,309.556,-158.159,168.976,54.429,160.474
C06095=1005.498,309.197,-158.115,168.966,54.437,160.473
C06096=1005.491,308.837,-158.070,168.956,54.445,160.473
C06097=1005.484,308.479,-158.025,168.947,54.453,160.473
C06098=1005.480,308.239,-157.995,168.940,54.458,160.472
C06099=1005.475,308.000,-157.966,168.933,54.464,160.472
C06100=1005.471,307.762,-157.937,168.926,54.470,160.472
C06101=1005.465,307.522,-157.908,168.920,54.475,160.472
C06102=1005.461,307.284,-157.878,168.913,54.481,160.471
C06103=1005.456,307.045,-157.849,168.906,54.486,160.471
C06104=1005.452,306.806,-157.821,168.900,54.491,160.471
C06105=1005.447,306.567,-157.791,168.894,54.497,160.471
C06106=1005.202,307.081,-158.220,168.889,54.514,160.474
C06107=1005.209,307.438,-158.263,168.899,54.506,160.474
C06108=1005.217,307.795,-158.306,168.908,54.497,160.474
C06109=1005.223,308.152,-158.350,168.919,54.490,160.475
C06110=1005.229,308.509,-158.395,168.928,54.482,160.475
C06111=1005.236,308.870,-158.439,168.938,54.473,160.475
C06112=1005.243,309.231,-158.485,168.948,54.466,160.476
C06113=1005.250,309.593,-158.530,168.959,54.457,160.476
C06114=1005.256,309.954,-158.575,168.969,54.449,160.477
C06115=1005.261,310.203,-158.605,168.975,54.443,160.477
C06116=1005.266,310.451,-158.636,168.983,54.438,160.477
C06117=1005.271,310.698,-158.666,168.989,54.432,160.478
C06118=1005.276,310.946,-158.697,168.996,54.427,160.478
C06119=1005.280,311.195,-158.729,169.004,54.421,160.478
C06120=1005.285,311.442,-158.760,169.010,54.416,160.479
C06121=1005.290,311.690,-158.790,169.018,54.410,160.479
C06122=1005.295,311.938,-158.821,169.025,54.405,160.479
C06123=1005.300,312.186,-158.853,169.032,54.399,160.480
C06124=1005.304,312.434,-158.884,169.039,54.394,160.480
C06125=1005.309,312.682,-158.915,169.045,54.389,160.480
C06126=1005.314,312.930,-158.946,169.053,54.383,160.481
C06127=1005.319,313.178,-158.977,169.060,54.378,160.481
C06128=1005.324,313.426,-159.008,169.067,54.372,160.481
C06129=1005.329,313.674,-159.039,169.074,54.367,160.481
C06130=1005.333,313.922,-159.071,169.082,54.361,160.482
C06131=1005.338,314.170,-159.102,169.088,54.356,160.482
C06132=1005.344,314.418,-159.133,169.096,54.350,160.483
C06133=1005.349,314.666,-159.164,169.103,54.345,160.483
C06134=1005.354,314.913,-159.195,169.110,54.339,160.483
C06135=1005.358,315.162,-159.227,169.117,54.334,160.483
C06136=1005.363,315.410,-159.258,169.124,54.328,160.484
C06137=1005.369,315.658,-159.289,169.131,54.323,160.484
C06138=1005.374,315.906,-159.320,169.139,54.317,160.484
C06139=1005.379,316.154,-159.351,169.145,54.312,160.485
C06140=1005.384,316.401,-159.383,169.153,54.306,160.485
C06141=1005.389,316.650,-159.415,169.160,54.301,160.486
C06142=1005.394,316.898,-159.446,169.168,54.296,160.486
C06143=1005.399,317.145,-159.477,169.174,54.290,160.486
C06144=1005.404,317.394,-159.508,169.182,54.285,160.487
C06145=1005.410,317.641,-159.540,169.189,54.279,160.487
C06146=1005.414,317.889,-159.571,169.196,54.274,160.487
C06147=1005.419,318.137,-159.603,169.203,54.269,160.488
C06148=1005.424,318.385,-159.634,169.211,54.263,160.488
C06149=1005.430,318.633,-159.666,169.219,54.258,160.489
C06150=1005.435,318.880,-159.697,169.225,54.252,160.489
C06151=1005.441,319.129,-159.729,169.233,54.247,160.489
C06152=1005.446,319.377,-159.761,169.240,54.242,160.490
C06153=1005.451,319.625,-159.792,169.248,54.236,160.490
C06154=1005.456,319.872,-159.823,169.254,54.231,160.490
C06155=1005.461,320.120,-159.855,169.262,54.226,160.491
C06156=1005.467,320.369,-159.886,169.270,54.220,160.491
C06157=1005.472,320.617,-159.919,169.277,54.215,160.492
C06158=1005.477,320.864,-159.950,169.285,54.210,160.492
C06159=1005.482,321.112,-159.982,169.291,54.205,160.492
C06160=1005.488,321.360,-160.013,169.299,54.199,160.493
C06161=1005.494,321.608,-160.045,169.307,54.194,160.493
C06162=1005.499,321.855,-160.077,169.314,54.189,160.494
C06163=1005.504,322.103,-160.109,169.322,54.184,160.494
C06164=1005.510,322.352,-160.141,169.328,54.179,160.495
C06165=1005.515,322.600,-160.172,169.336,54.173,160.495
C06166=1005.521,322.848,-160.204,169.344,54.168,160.496
C06167=1005.526,323.095,-160.236,169.351,54.163,160.496
C06168=1005.531,323.343,-160.268,169.359,54.158,160.496
C06169=1005.537,323.591,-160.300,169.367,54.152,160.497
C06170=1005.542,323.839,-160.331,169.374,54.147,160.497
C06171=1005.547,324.070,-160.362,169.380,54.142,160.497
C06172=1005.553,324.302,-160.391,169.387,54.137,160.498
C06173=1005.558,324.534,-160.421,169.395,54.132,160.499
C06174=1005.563,324.766,-160.452,169.402,54.127,160.499
C06175=1005.567,324.996,-160.482,169.409,54.123,160.499
C06176=1005.572,325.228,-160.512,169.416,54.118,160.500
C06177=1005.577,325.459,-160.542,169.423,54.113,160.500
C06178=1005.582,325.692,-160.573,169.430,54.108,160.501
C06179=1005.588,325.939,-160.605,169.438,54.103,160.501
C06180=1005.593,326.187,-160.638,169.445,54.099,160.502
C06181=1005.598,326.435,-160.671,169.453,54.093,160.502
C06182=1005.604,326.683,-160.702,169.461,54.088,160.503
C06183=1005.609,326.931,-160.735,169.468,54.083,160.503
C06184=1005.614,327.178,-160.768,169.476,54.078,160.503
C06185=1005.620,327.427,-160.800,169.484,54.073,160.504
C06186=1005.625,327.674,-160.833,169.491,54.068,160.505
C06187=1005.630,327.922,-160.866,169.499,54.062,160.505
C06188=1005.636,328.170,-160.898,169.507,54.057,160.506
C06189=1005.641,328.417,-160.931,169.514,54.053,160.506
C06190=1005.647,328.665,-160.963,169.522,54.048,160.507
C06191=1005.653,328.913,-160.997,169.530,54.042,160.507
C06192=1005.658,329.161,-161.029,169.538,54.037,160.508
C06193=1005.664,329.409,-161.062,169.545,54.033,160.508
C06194=1005.669,329.657,-161.095,169.553,54.028,160.509
C06195=1005.674,329.904,-161.127,169.560,54.022,160.509
C06196=1005.680,330.152,-161.160,169.569,54.017,160.510
C06197=1005.686,330.400,-161.193,169.576,54.012,160.510
C06198=1005.691,330.648,-161.227,169.584,54.007,160.511
C06199=1005.697,330.895,-161.259,169.592,54.002,160.511
C06200=1005.703,331.143,-161.293,169.600,53.997,160.512
C06201=1005.708,331.391,-161.325,169.607,53.993,160.512
C06202=1005.713,331.639,-161.358,169.615,53.988,160.513
C06203=1005.719,331.887,-161.392,169.623,53.983,160.514
C06204=1005.724,332.134,-161.425,169.631,53.978,160.514
C06205=1005.730,332.381,-161.459,169.638,53.973,160.514
C06206=1005.735,332.629,-161.492,169.646,53.968,160.515
C06207=1005.741,332.877,-161.526,169.654,53.963,160.515
C06208=1005.747,333.125,-161.558,169.662,53.958,160.516
C06209=1005.753,333.373,-161.592,169.669,53.953,160.517
C06210=1005.758,333.621,-161.625,169.678,53.949,160.517
C06211=1005.763,333.868,-161.658,169.686,53.944,160.518
C06212=1005.769,334.116,-161.691,169.694,53.939,160.519
C06213=1005.775,334.363,-161.725,169.702,53.934,160.519
C06214=1005.780,334.611,-161.759,169.709,53.929,160.520
C06215=1005.786,334.859,-161.792,169.718,53.924,160.520
C06216=1005.791,335.107,-161.825,169.726,53.919,160.521
C06217=1005.798,335.354,-161.859,169.734,53.914,160.521
C06218=1005.804,335.602,-161.892,169.742,53.909,160.522
C06219=1005.495,333.430,-161.961,169.654,53.985,160.521
C06220=1005.490,333.182,-161.928,169.646,53.990,160.520
C06221=1005.484,332.934,-161.894,169.638,53.994,160.520
C06222=1005.478,332.687,-161.861,169.630,53.999,160.519
C06223=1005.472,332.439,-161.828,169.622,54.004,160.518
C06224=1005.468,332.191,-161.795,169.614,54.009,160.518
C06225=1005.462,331.944,-161.762,169.607,54.014,160.517
C06226=1005.456,331.696,-161.728,169.599,54.019,160.517
C06227=1005.451,331.448,-161.695,169.591,54.024,160.516
C06228=1005.446,331.201,-161.662,169.583,54.029,160.515
C06229=1005.440,330.953,-161.629,169.576,54.033,160.515
C06230=1005.435,330.705,-161.595,169.568,54.038,160.514
C06231=1005.429,330.457,-161.563,169.559,54.043,160.514
C06232=1005.424,330.209,-161.530,169.551,54.048,160.513
C06233=1005.418,329.961,-161.497,169.544,54.053,160.513
C06234=1005.412,329.714,-161.464,169.537,54.058,160.512
C06235=1005.407,329.466,-161.432,169.528,54.063,160.512
C06236=1005.401,329.218,-161.399,169.521,54.068,160.511
C06237=1005.396,328.970,-161.367,169.513,54.073,160.511
C06238=1005.391,328.723,-161.334,169.505,54.078,160.510
C06239=1005.385,328.475,-161.301,169.497,54.083,160.509
C06240=1005.379,328.227,-161.268,169.490,54.088,160.509
C06241=1005.374,327.979,-161.235,169.482,54.093,160.509
C06242=1005.368,327.731,-161.203,169.474,54.098,160.508
C06243=1005.363,327.484,-161.170,169.467,54.103,160.508
C06244=1005.358,327.235,-161.138,169.459,54.108,160.507
C06245=1005.353,326.989,-161.105,169.451,54.114,160.507
C06246=1005.347,326.740,-161.073,169.444,54.118,160.506
C06247=1005.342,326.493,-161.041,169.436,54.123,160.505
C06248=1005.336,326.245,-161.008,169.428,54.129,160.505
C06249=1005.332,325.997,-160.976,169.421,54.133,160.505
C06250=1005.326,325.749,-160.944,169.413,54.138,160.504
C06251=1005.321,325.501,-160.911,169.407,54.144,160.504
C06252=1005.312,325.096,-160.858,169.393,54.152,160.503
C06253=1005.303,324.690,-160.805,169.381,54.160,160.502
C06254=1005.294,324.285,-160.752,169.369,54.169,160.501
C06255=1005.286,323.879,-160.700,169.356,54.177,160.500
C06256=1005.281,323.631,-160.668,169.350,54.182,160.500
C06257=1005.275,323.383,-160.636,169.342,54.187,160.500
C06258=1005.269,323.135,-160.605,169.334,54.193,160.499
C06259=1005.265,322.888,-160.572,169.327,54.198,160.499
C06260=1005.259,322.639,-160.540,169.319,54.203,160.498
C06261=1005.253,322.392,-160.509,169.311,54.208,160.498
C06262=1005.248,322.144,-160.477,169.305,54.214,160.497
C06263=1005.243,321.896,-160.446,169.296,54.219,160.497
C06264=1005.238,321.648,-160.414,169.290,54.224,160.497
C06265=1005.232,321.400,-160.382,169.282,54.229,160.496
C06266=1005.227,321.153,-160.350,169.274,54.235,160.496
C06267=1005.221,320.904,-160.319,169.267,54.240,160.495
C06268=1005.216,320.656,-160.287,169.259,54.245,160.495
C06269=1005.210,320.409,-160.256,169.253,54.250,160.494
C06270=1005.206,320.160,-160.224,169.245,54.255,160.494
C06271=1005.201,319.913,-160.192,169.238,54.260,160.494
C06272=1005.195,319.665,-160.161,169.230,54.266,160.493
C06273=1005.190,319.416,-160.129,169.223,54.271,160.493
C06274=1005.184,319.169,-160.098,169.216,54.276,160.492
C06275=1005.180,318.920,-160.066,169.208,54.282,160.492
C06276=1005.174,318.673,-160.035,169.201,54.287,160.491
C06277=1005.169,318.425,-160.004,169.193,54.292,160.491
C06278=1005.164,318.177,-159.972,169.187,54.298,160.491
C06279=1005.159,317.929,-159.941,169.178,54.303,160.490
C06280=1005.154,317.682,-159.909,169.172,54.308,160.490
C06281=1005.149,317.433,-159.878,169.164,54.314,160.489
C06282=1005.144,317.186,-159.846,169.158,54.319,160.489
C06283=1005.139,316.938,-159.815,169.149,54.324,160.489
C06284=1005.133,316.663,-159.781,169.142,54.330,160.488
C06285=1005.127,316.389,-159.746,169.135,54.336,160.488
C06286=1005.122,316.115,-159.711,169.126,54.342,160.488
C06287=1005.116,315.841,-159.677,169.118,54.348,160.487
C06288=1005.111,315.593,-159.646,169.111,54.354,160.487
C06289=1005.106,315.345,-159.615,169.104,54.358,160.486
C06290=1005.101,315.097,-159.582,169.096,54.364,160.486
C06291=1005.096,314.849,-159.551,169.089,54.369,160.486
C06292=1005.092,314.601,-159.521,169.082,54.375,160.485
C06293=1005.087,314.353,-159.490,169.075,54.380,160.485
C06294=1005.081,314.106,-159.458,169.068,54.386,160.485
C06295=1005.077,313.857,-159.427,169.061,54.391,160.484
C06296=1005.072,313.609,-159.396,169.054,54.397,160.484
C06297=1005.067,313.361,-159.365,169.047,54.402,160.484
C06298=1005.062,313.113,-159.334,169.039,54.407,160.483
C06299=1005.057,312.865,-159.303,169.032,54.413,160.483
C06300=1005.053,312.617,-159.272,169.025,54.418,160.482
C06301=1005.048,312.369,-159.241,169.019,54.423,160.482
C06302=1005.043,312.121,-159.210,169.011,54.429,160.482
C06303=1005.038,311.873,-159.179,169.004,54.434,160.481
C06304=1005.033,311.625,-159.148,168.997,54.440,160.481
C06305=1005.028,311.377,-159.117,168.990,54.445,160.481
C06306=1005.024,311.129,-159.086,168.983,54.451,160.480
C06307=1005.019,310.881,-159.055,168.976,54.456,160.480
C06308=1005.014,310.633,-159.024,168.969,54.462,160.480
C06309=1005.010,310.386,-158.994,168.962,54.467,160.479
C06310=1005.005,310.137,-158.963,168.955,54.473,160.479
C06311=1005.001,309.890,-158.932,168.949,54.479,160.479
C06312=1004.994,309.552,-158.890,168.939,54.486,160.479
C06313=1004.988,309.214,-158.848,168.929,54.494,160.478
C06314=1004.981,308.876,-158.806,168.920,54.501,160.478
C06315=1004.975,308.539,-158.764,168.910,54.508,160.477
C06316=1004.971,308.300,-158.734,168.903,54.514,160.477
C06317=1004.966,308.060,-158.705,168.897,54.520,160.477
C06318=1004.962,307.821,-158.675,168.891,54.525,160.477
C06319=1004.957,307.581,-158.646,168.884,54.530,160.476
C06320=1004.711,308.068,-159.071,168.880,54.545,160.479
C06321=1004.716,308.319,-159.102,168.886,54.540,160.479
C06322=1004.720,308.570,-159.134,168.893,54.535,160.479
C06323=1004.727,308.936,-159.179,168.903,54.526,160.480
C06324=1004.734,309.302,-159.224,168.914,54.518,160.480
C06325=1004.741,309.668,-159.270,168.923,54.510,160.481
C06326=1004.748,310.034,-159.315,168.935,54.502,160.481
C06327=1004.753,310.282,-159.346,168.941,54.497,160.482
C06328=1004.757,310.530,-159.377,168.948,54.491,160.482
C06329=1004.762,310.778,-159.408,168.955,54.486,160.482
C06330=1004.766,311.026,-159.438,168.962,54.480,160.483
C06331=1004.771,311.274,-159.469,168.969,54.475,160.483
C06332=1004.776,311.522,-159.500,168.976,54.469,160.483
C06333=1004.780,311.770,-159.531,168.983,54.464,160.483
C06334=1004.786,312.018,-159.562,168.990,54.459,160.484
C06335=1004.791,312.266,-159.593,168.997,54.453,160.484
C06336=1004.794,312.514,-159.624,169.004,54.448,160.484
C06337=1004.799,312.762,-159.655,169.011,54.442,160.485
C06338=1004.805,313.010,-159.686,169.018,54.437,160.485
C06339=1004.810,313.258,-159.717,169.025,54.432,160.486
C06340=1004.814,313.505,-159.748,169.033,54.426,160.486
C06341=1004.819,313.754,-159.780,169.039,54.421,160.486
C06342=1004.824,314.002,-159.811,169.047,54.415,160.487
C06343=1004.829,314.250,-159.841,169.054,54.410,160.487
C06344=1004.834,314.498,-159.872,169.060,54.405,160.487
C06345=1004.839,314.746,-159.903,169.069,54.400,160.488
C06346=1004.843,314.994,-159.935,169.075,54.394,160.488
C06347=1004.848,315.241,-159.966,169.083,54.389,160.489
C06348=1004.853,315.489,-159.997,169.089,54.383,160.489
C06349=1004.858,315.738,-160.028,169.097,54.378,160.489
C06350=1004.863,315.986,-160.059,169.104,54.373,160.490
C06351=1004.869,316.233,-160.091,169.111,54.368,160.490
C06352=1004.873,316.482,-160.122,169.118,54.362,160.490
C06353=1004.878,316.730,-160.153,169.125,54.357,160.491
C06354=1004.884,316.977,-160.185,169.133,54.352,160.491
C06355=1004.889,317.225,-160.216,169.140,54.346,160.492
C06356=1004.894,317.474,-160.247,169.147,54.341,160.492
C06357=1004.898,317.721,-160.279,169.155,54.336,160.493
C06358=1004.904,317.970,-160.310,169.162,54.330,160.493
C06359=1004.909,318.217,-160.342,169.169,54.325,160.493
C06360=1004.914,318.465,-160.373,169.177,54.320,160.494
C06361=1004.919,318.713,-160.404,169.184,54.315,160.494
C06362=1004.924,318.961,-160.436,169.191,54.309,160.494
C06363=1004.929,319.209,-160.467,169.198,54.305,160.495
C06364=1004.934,319.457,-160.498,169.206,54.299,160.495
C06365=1004.940,319.704,-160.530,169.213,54.294,160.496
C06366=1004.945,319.952,-160.561,169.221,54.289,160.496
C06367=1004.951,320.201,-160.593,169.228,54.284,160.497
C06368=1004.955,320.449,-160.625,169.235,54.278,160.497
C06369=1004.960,320.697,-160.656,169.242,54.273,160.497
C06370=1004.966,320.944,-160.688,169.250,54.268,160.498
C06371=1004.971,321.192,-160.719,169.258,54.262,160.498
C06372=1004.977,321.440,-160.751,169.265,54.258,160.499
C06373=1004.981,321.688,-160.783,169.273,54.252,160.499
C06374=1004.987,321.936,-160.815,169.280,54.247,160.500
C06375=1004.992,322.184,-160.846,169.287,54.242,160.500
C06376=1004.998,322.432,-160.878,169.294,54.237,160.501
C06377=1005.003,322.680,-160.909,169.302,54.231,160.501
C06378=1005.009,322.927,-160.941,169.310,54.226,160.502
C06379=1005.013,323.176,-160.973,169.317,54.222,160.502
C06380=1005.019,323.424,-161.005,169.325,54.216,160.503
C06381=1005.024,323.671,-161.036,169.332,54.211,160.503
C06382=1005.030,323.920,-161.068,169.340,54.206,160.503
C06383=1005.037,324.267,-161.113,169.350,54.199,160.504
C06384=1005.045,324.615,-161.158,169.361,54.192,160.505
C06385=1005.052,324.963,-161.204,169.372,54.185,160.506
C06386=1005.060,325.311,-161.249,169.382,54.177,160.506
C06387=1005.065,325.558,-161.282,169.390,54.172,160.507
C06388=1005.071,325.806,-161.314,169.397,54.168,160.507
C06389=1005.075,326.054,-161.346,169.405,54.162,160.508
C06390=1005.080,326.303,-161.379,169.413,54.157,160.508
C06391=1005.086,326.550,-161.411,169.420,54.152,160.509
C06392=1005.091,326.797,-161.443,169.428,54.147,160.509
C06393=1005.096,327.045,-161.477,169.436,54.142,160.510
C06394=1005.102,327.293,-161.508,169.443,54.137,160.510
C06395=1005.107,327.541,-161.541,169.451,54.132,160.511
C06396=1005.113,327.789,-161.574,169.459,54.127,160.511
C06397=1005.118,328.037,-161.606,169.466,54.123,160.512
C06398=1005.123,328.285,-161.639,169.474,54.118,160.513
C06399=1005.129,328.532,-161.671,169.481,54.113,160.513
C06400=1005.134,328.780,-161.704,169.489,54.107,160.513
C06401=1005.139,329.028,-161.736,169.497,54.102,160.514
C06402=1005.145,329.276,-161.769,169.505,54.097,160.515
C06403=1005.151,329.524,-161.802,169.512,54.093,160.515
C06404=1005.156,329.771,-161.835,169.520,54.088,160.516
C06405=1005.162,330.019,-161.867,169.528,54.083,160.516
C06406=1005.167,330.267,-161.900,169.536,54.078,160.517
C06407=1005.172,330.515,-161.933,169.544,54.073,160.517
C06408=1005.178,330.762,-161.966,169.552,54.068,160.518
C06409=1005.184,331.010,-161.999,169.559,54.064,160.519
C06410=1005.189,331.258,-162.031,169.567,54.059,160.519
C06411=1004.884,329.077,-162.106,169.480,54.131,160.517
C06412=1004.877,328.829,-162.073,169.473,54.136,160.517
C06413=1004.873,328.581,-162.041,169.465,54.141,160.516
C06414=1004.867,328.333,-162.007,169.457,54.146,160.516
C06415=1004.862,328.086,-161.976,169.450,54.151,160.515
C06416=1004.856,327.838,-161.942,169.442,54.156,160.515
C06417=1004.851,327.590,-161.910,169.435,54.160,160.514
C06418=1004.845,327.342,-161.878,169.427,54.165,160.513
C06419=1004.840,327.095,-161.845,169.419,54.170,160.513
C06420=1004.835,326.846,-161.813,169.412,54.175,160.512
C06421=1004.830,326.599,-161.781,169.404,54.180,160.512
C06422=1004.824,326.351,-161.748,169.396,54.186,160.511
C06423=1004.820,326.103,-161.715,169.389,54.190,160.511
C06424=1004.814,325.855,-161.684,169.381,54.195,160.510
C06425=1004.809,325.607,-161.650,169.374,54.200,160.510
C06426=1004.803,325.360,-161.619,169.366,54.205,160.509
C06427=1004.799,325.112,-161.586,169.359,54.210,160.509
C06428=1004.792,324.824,-161.548,169.350,54.216,160.508
C06429=1004.787,324.536,-161.511,169.341,54.222,160.508
C06430=1004.780,324.247,-161.473,169.333,54.228,160.507
C06431=1004.774,323.959,-161.437,169.323,54.233,160.506
C06432=1004.769,323.712,-161.405,169.316,54.239,160.506
C06433=1004.763,323.463,-161.373,169.309,54.244,160.505
C06434=1004.758,323.216,-161.341,169.300,54.249,160.505
C06435=1004.753,322.968,-161.309,169.293,54.254,160.504
C06436=1004.747,322.719,-161.278,169.286,54.259,160.504
C06437=1004.742,322.472,-161.246,169.278,54.264,160.503
C06438=1004.737,322.224,-161.215,169.271,54.269,160.503
C06439=1004.731,321.977,-161.183,169.263,54.274,160.502
C06440=1004.725,321.728,-161.152,169.256,54.280,160.502
C06441=1004.721,321.480,-161.119,169.248,54.285,160.501
C06442=1004.715,321.233,-161.088,169.241,54.289,160.501
C06443=1004.710,320.984,-161.057,169.233,54.295,160.501
C06444=1004.705,320.737,-161.025,169.226,54.299,160.500
C06445=1004.700,320.489,-160.994,169.219,54.305,160.500
C06446=1004.695,320.240,-160.962,169.212,54.310,160.499
C06447=1004.690,319.992,-160.931,169.204,54.315,160.499
C06448=1004.684,319.745,-160.899,169.197,54.320,160.498
C06449=1004.679,319.497,-160.867,169.189,54.326,160.498
C06450=1004.674,319.249,-160.836,169.182,54.330,160.497
C06451=1004.669,319.001,-160.805,169.174,54.336,160.497
C06452=1004.664,318.753,-160.773,169.168,54.341,160.497
C06453=1004.659,318.505,-160.742,169.160,54.346,160.496
C06454=1004.654,318.257,-160.711,169.153,54.352,160.496
C06455=1004.648,318.009,-160.680,169.145,54.357,160.495
C06456=1004.643,317.762,-160.648,169.138,54.362,160.495
C06457=1004.639,317.513,-160.616,169.130,54.367,160.494
C06458=1004.634,317.265,-160.585,169.124,54.372,160.494
C06459=1004.628,317.018,-160.554,169.116,54.378,160.494
C06460=1004.623,316.770,-160.523,169.109,54.383,160.493
C06461=1004.618,316.521,-160.492,169.101,54.388,160.493
C06462=1004.614,316.273,-160.460,169.095,54.394,160.492
C06463=1004.608,316.025,-160.429,169.087,54.398,160.492
C06464=1004.603,315.777,-160.398,169.080,54.404,160.491
C06465=1004.599,315.530,-160.367,169.073,54.409,160.491
C06466=1004.594,315.282,-160.336,169.065,54.414,160.491
C06467=1004.589,315.034,-160.304,169.058,54.420,160.490
C06468=1004.584,314.786,-160.273,169.052,54.425,160.490
C06469=1004.579,314.538,-160.242,169.044,54.431,160.490
C06470=1004.574,314.290,-160.211,169.037,54.435,160.489
C06471=1004.569,314.042,-160.181,169.029,54.441,160.489
C06472=1004.564,313.794,-160.150,169.023,54.446,160.488
C06473=1004.560,313.546,-160.118,169.016,54.452,160.488
C06474=1004.555,313.297,-160.087,169.008,54.457,160.488
C06475=1004.550,313.050,-160.057,169.001,54.462,160.487
C06476=1004.545,312.802,-160.026,168.995,54.467,160.487
C06477=1004.540,312.554,-159.995,168.987,54.473,160.487
C06478=1004.536,312.306,-159.963,168.980,54.478,160.486
C06479=1004.531,312.058,-159.933,168.973,54.484,160.486
C06480=1004.526,311.810,-159.902,168.966,54.489,160.485
C06481=1004.522,311.562,-159.871,168.959,54.494,160.485
C06482=1004.517,311.314,-159.840,168.951,54.500,160.485
C06483=1004.512,311.066,-159.808,168.945,54.505,160.484
C06484=1004.508,310.818,-159.778,168.938,54.510,160.484
C06485=1004.503,310.570,-159.748,168.931,54.516,160.484
C06486=1004.499,310.322,-159.717,168.924,54.521,160.483
C06487=1004.494,310.074,-159.686,168.917,54.527,160.483
C06488=1004.487,309.706,-159.640,168.906,54.535,160.482
C06489=1004.480,309.337,-159.595,168.896,54.543,160.482
C06490=1004.474,308.969,-159.549,168.886,54.551,160.481
C06491=1004.466,308.572,-159.500,168.876,54.559,160.481
C06492=1004.220,309.003,-159.920,168.869,54.574,160.483
C06493=1004.225,309.281,-159.953,168.877,54.568,160.483
C06494=1004.229,309.558,-159.988,168.884,54.562,160.484
C06495=1004.235,309.836,-160.022,168.893,54.556,160.484
C06496=1004.240,310.113,-160.056,168.901,54.550,160.485
C06497=1004.245,310.362,-160.088,168.907,54.545,160.485
C06498=1004.249,310.610,-160.118,168.915,54.539,160.485
C06499=1004.254,310.858,-160.149,168.921,54.534,160.486
C06500=1004.258,311.106,-160.179,168.928,54.529,160.486
C06501=1004.263,311.354,-160.210,168.935,54.523,160.486
C06502=1004.268,311.602,-160.242,168.943,54.518,160.487
C06503=1004.272,311.850,-160.272,168.949,54.513,160.487
C06504=1004.277,312.098,-160.303,168.956,54.508,160.487
C06505=1004.281,312.346,-160.333,168.964,54.502,160.488
C06506=1004.286,312.594,-160.364,168.971,54.497,160.488
C06507=1004.291,312.842,-160.396,168.977,54.492,160.489
C06508=1004.296,313.090,-160.427,168.985,54.486,160.489
C06509=1004.300,313.338,-160.457,168.992,54.481,160.489
C06510=1004.305,313.586,-160.488,168.999,54.476,160.490
C06511=1004.311,313.834,-160.519,169.007,54.471,160.490
C06512=1004.315,314.082,-160.550,169.013,54.465,160.491
C06513=1004.319,314.330,-160.581,169.020,54.460,160.491
C06514=1004.324,314.578,-160.612,169.028,54.455,160.492
C06515=1004.330,314.826,-160.644,169.035,54.450,160.492
C06516=1004.335,315.074,-160.675,169.042,54.444,160.492
C06517=1004.339,315.321,-160.705,169.049,54.439,160.493
C06518=1004.344,315.570,-160.737,169.056,54.434,160.493
C06519=1004.349,315.818,-160.768,169.064,54.428,160.493
C06520=1004.354,316.066,-160.799,169.071,54.424,160.494
C06521=1004.359,316.313,-160.830,169.077,54.418,160.494
C06522=1004.364,316.562,-160.861,169.085,54.413,160.495
C06523=1004.368,316.809,-160.892,169.092,54.408,160.495
C06524=1004.373,317.057,-160.923,169.100,54.402,160.496
C06525=1004.379,317.305,-160.955,169.107,54.398,160.496
C06526=1004.384,317.553,-160.986,169.114,54.392,160.496
C06527=1004.389,317.801,-161.017,169.122,54.387,160.497
C06528=1004.393,318.049,-161.049,169.128,54.382,160.497
C06529=1004.398,318.297,-161.080,169.136,54.377,160.498
C06530=1004.404,318.545,-161.111,169.143,54.372,160.498
C06531=1004.409,318.793,-161.143,169.151,54.367,160.499
C06532=1004.414,319.041,-161.174,169.158,54.361,160.499
C06533=1004.419,319.288,-161.205,169.166,54.356,160.500
C06534=1004.424,319.537,-161.237,169.172,54.351,160.500
C06535=1004.429,319.785,-161.268,169.181,54.346,160.501
C06536=1004.434,320.033,-161.300,169.187,54.341,160.501
C06537=1004.439,320.281,-161.330,169.195,54.336,160.502
C06538=1004.445,320.529,-161.362,169.202,54.331,160.502
C06539=1004.450,320.777,-161.395,169.209,54.326,160.502
C06540=1004.455,321.025,-161.426,169.217,54.321,160.503
C06541=1004.460,321.272,-161.457,169.224,54.315,160.503
C06542=1004.465,321.520,-161.488,169.232,54.310,160.504
C06543=1004.471,321.768,-161.520,169.240,54.305,160.505
C06544=1004.476,322.017,-161.553,169.247,54.300,160.505
C06545=1004.481,322.265,-161.584,169.255,54.295,160.505
C06546=1004.487,322.512,-161.615,169.262,54.290,160.506
C06547=1004.492,322.760,-161.647,169.270,54.285,160.506
C06548=1004.498,323.009,-161.678,169.277,54.280,160.507
C06549=1004.503,323.256,-161.710,169.285,54.275,160.507
C06550=1004.508,323.504,-161.742,169.291,54.270,160.508
C06551=1004.513,323.751,-161.774,169.300,54.265,160.508
C06552=1004.519,324.000,-161.805,169.307,54.260,160.509
C06553=1004.524,324.237,-161.836,169.315,54.255,160.510
C06554=1004.528,324.475,-161.866,169.322,54.251,160.510
C06555=1004.534,324.713,-161.898,169.328,54.245,160.510
C06556=1004.538,324.950,-161.928,169.336,54.241,160.511
C06557=1004.544,325.188,-161.959,169.343,54.236,160.511
C06558=1004.548,325.425,-161.990,169.350,54.231,160.512
C06559=1004.554,325.663,-162.021,169.358,54.226,160.512
C06560=1004.558,325.901,-162.052,169.365,54.222,160.513
C06561=1004.564,326.149,-162.085,169.372,54.217,160.513
C06562=1004.569,326.396,-162.117,169.380,54.212,160.514
C06563=1004.574,326.644,-162.149,169.388,54.207,160.515
C06564=1004.580,326.892,-162.181,169.396,54.203,160.515
C06565=1004.277,324.708,-162.260,169.311,54.272,160.513
C06566=1004.270,324.374,-162.217,169.301,54.278,160.512
C06567=1004.263,324.040,-162.174,169.291,54.285,160.511
C06568=1004.258,323.792,-162.143,169.283,54.290,160.511
C06569=1004.253,323.544,-162.110,169.276,54.295,160.510
C06570=1004.248,323.296,-162.079,169.268,54.300,160.510
C06571=1004.242,323.048,-162.047,169.261,54.305,160.509
C06572=1004.237,322.800,-162.016,169.253,54.310,160.509
C06573=1004.231,322.553,-161.984,169.246,54.315,160.508
C06574=1004.226,322.305,-161.952,169.238,54.320,160.508
C06575=1004.221,322.057,-161.921,169.231,54.325,160.507
C06576=1004.215,321.808,-161.889,169.223,54.330,160.506
C06577=1004.210,321.560,-161.858,169.216,54.335,160.506
C06578=1004.205,321.313,-161.826,169.208,54.340,160.506
C06579=1004.200,321.065,-161.795,169.201,54.345,160.505
C06580=1004.195,320.817,-161.763,169.193,54.351,160.505
C06581=1004.190,320.569,-161.731,169.186,54.355,160.504
C06582=1004.185,320.321,-161.700,169.178,54.360,160.503
C06583=1004.179,320.074,-161.669,169.171,54.366,160.503
C06584=1004.174,319.825,-161.638,169.163,54.371,160.503
C06585=1004.170,319.577,-161.606,169.157,54.376,160.502
C06586=1004.165,319.330,-161.575,169.150,54.380,160.502
C06587=1004.159,319.081,-161.544,169.141,54.386,160.501
C06588=1004.154,318.834,-161.512,169.135,54.391,160.501
C06589=1004.149,318.586,-161.481,169.127,54.396,160.500
C06590=1004.145,318.337,-161.450,169.120,54.401,160.500
C06591=1004.139,318.090,-161.418,169.112,54.406,160.499
C06592=1004.134,317.842,-161.387,169.105,54.411,160.499
C06593=1004.129,317.594,-161.356,169.098,54.416,160.498
C06594=1004.124,317.346,-161.324,169.091,54.422,160.498
C06595=1004.119,317.098,-161.293,169.083,54.426,160.498
C06596=1004.114,316.849,-161.262,169.076,54.432,160.497
C06597=1004.109,316.601,-161.231,169.069,54.437,160.497
C06598=1004.104,316.353,-161.200,169.062,54.442,160.496
C06599=1004.099,316.106,-161.169,169.054,54.447,160.496
C06600=1004.094,315.858,-161.138,169.047,54.452,160.495
C06601=1004.090,315.610,-161.106,169.040,54.457,160.495
C06602=1004.085,315.362,-161.075,169.033,54.463,160.494
C06603=1004.080,315.114,-161.044,169.025,54.467,160.494
C06604=1004.075,314.865,-161.013,169.019,54.473,160.494
C06605=1004.070,314.618,-160.983,169.011,54.478,160.493
C06606=1004.066,314.370,-160.951,169.004,54.483,160.493
C06607=1004.061,314.121,-160.920,168.997,54.488,160.492
C06608=1004.056,313.874,-160.890,168.990,54.494,160.492
C06609=1004.051,313.626,-160.859,168.983,54.499,160.491
C06610=1004.046,313.378,-160.828,168.976,54.504,160.491
C06611=1004.042,313.130,-160.797,168.968,54.510,160.491
C06612=1004.037,312.882,-160.766,168.961,54.514,160.490
C06613=1004.032,312.634,-160.735,168.955,54.520,160.490
C06614=1004.028,312.386,-160.704,168.947,54.526,160.490
C06615=1004.023,312.138,-160.673,168.940,54.530,160.489
C06616=1004.018,311.890,-160.642,168.933,54.535,160.489
C06617=1004.014,311.642,-160.612,168.926,54.541,160.488
C06618=1004.009,311.393,-160.581,168.919,54.547,160.488
C06619=1004.005,311.146,-160.550,168.912,54.551,160.487
C06620=1004.001,310.934,-160.524,168.906,54.556,160.487
C06621=1003.996,310.722,-160.498,168.900,54.560,160.487
C06622=1003.993,310.510,-160.471,168.894,54.565,160.486
C06623=1003.989,310.298,-160.445,168.888,54.569,160.486
C06624=1003.985,310.087,-160.419,168.882,54.574,160.486
C06625=1003.981,309.874,-160.393,168.877,54.579,160.486
C06626=1003.977,309.663,-160.367,168.871,54.583,160.485
C06627=1003.974,309.451,-160.341,168.864,54.587,160.485
C06628=1003.727,309.889,-160.760,168.858,54.600,160.487
C06629=1003.731,310.101,-160.786,168.866,54.596,160.487
C06630=1003.735,310.315,-160.812,168.872,54.591,160.487
C06631=1003.739,310.528,-160.839,168.877,54.586,160.488
C06632=1003.743,310.741,-160.866,168.883,54.582,160.488
C06633=1003.747,310.954,-160.891,168.890,54.578,160.488
C06634=1003.750,311.167,-160.919,168.895,54.573,160.489
C06635=1003.754,311.381,-160.945,168.901,54.569,160.489
C06636=1003.758,311.594,-160.971,168.907,54.565,160.489
C06637=1003.763,311.842,-161.002,168.914,54.559,160.490
C06638=1003.768,312.090,-161.033,168.922,54.553,160.490
C06639=1003.773,312.338,-161.064,168.929,54.549,160.491
C06640=1003.777,312.587,-161.094,168.935,54.543,160.491
C06641=1003.782,312.835,-161.125,168.942,54.539,160.492
C06642=1003.786,313.082,-161.156,168.950,54.533,160.492
C06643=1003.791,313.330,-161.187,168.957,54.528,160.492
C06644=1003.796,313.578,-161.218,168.964,54.523,160.493
C06645=1003.800,313.826,-161.249,168.972,54.517,160.493
C06646=1003.805,314.074,-161.280,168.979,54.513,160.494
C06647=1003.810,314.322,-161.311,168.985,54.507,160.494
C06648=1003.815,314.570,-161.341,168.992,54.502,160.494
C06649=1003.820,314.818,-161.372,169.000,54.497,160.495
C06650=1003.824,315.066,-161.404,169.007,54.492,160.495
C06651=1003.829,315.314,-161.435,169.014,54.487,160.496
C06652=1003.834,315.562,-161.465,169.021,54.481,160.496
C06653=1003.839,315.810,-161.496,169.029,54.477,160.497
C06654=1003.844,316.058,-161.527,169.035,54.472,160.497
C06655=1003.848,316.307,-161.559,169.043,54.466,160.498
C06656=1003.853,316.555,-161.590,169.050,54.461,160.498
C06657=1003.858,316.802,-161.621,169.057,54.457,160.499
C06658=1003.863,317.050,-161.652,169.065,54.451,160.499
C06659=1003.868,317.298,-161.683,169.072,54.446,160.499
C06660=1003.872,317.546,-161.714,169.080,54.441,160.500
C06661=1003.878,317.794,-161.745,169.087,54.436,160.500
C06662=1003.883,318.042,-161.777,169.094,54.431,160.501
C06663=1003.888,318.290,-161.808,169.101,54.425,160.501
C06664=1003.893,318.538,-161.839,169.108,54.421,160.502
C06665=1003.898,318.786,-161.871,169.116,54.416,160.502
C06666=1003.903,319.034,-161.902,169.123,54.411,160.503
C06667=1003.908,319.282,-161.933,169.130,54.406,160.503
C06668=1003.913,319.530,-161.965,169.138,54.401,160.504
C06669=1003.918,319.778,-161.996,169.145,54.396,160.504
C06670=1003.923,320.026,-162.027,169.153,54.391,160.505
C06671=1003.928,320.274,-162.059,169.160,54.386,160.505
C06672=1003.933,320.522,-162.090,169.167,54.381,160.506
C06673=1003.939,320.770,-162.121,169.175,54.376,160.506
C06674=1003.944,321.018,-162.152,169.182,54.371,160.507
C06675=1003.949,321.265,-162.184,169.190,54.365,160.507
C06676=1003.953,321.514,-162.216,169.197,54.361,160.508
C06677=1003.959,321.761,-162.247,169.205,54.356,160.508
C06678=1003.964,322.009,-162.278,169.212,54.351,160.509
C06679=1003.969,322.257,-162.310,169.220,54.345,160.509
C06680=1003.975,322.505,-162.342,169.227,54.341,160.510
C06681=1003.673,320.298,-162.426,169.144,54.408,160.507
C06682=1003.668,320.050,-162.395,169.136,54.413,160.506
C06683=1003.663,319.802,-162.363,169.129,54.419,160.506
C06684=1003.658,319.554,-162.332,169.122,54.423,160.506
C06685=1003.653,319.306,-162.300,169.114,54.428,160.505
C06686=1003.648,319.058,-162.269,169.107,54.433,160.504
C06687=1003.643,318.810,-162.238,169.099,54.439,160.504
C06688=1003.638,318.562,-162.207,169.092,54.443,160.503
C06689=1003.633,318.314,-162.175,169.085,54.448,160.503
C06690=1003.628,318.066,-162.144,169.077,54.454,160.502
C06691=1003.624,317.818,-162.113,169.070,54.458,160.502
C06692=1003.619,317.570,-162.082,169.063,54.463,160.501
C06693=1003.613,317.323,-162.051,169.056,54.469,160.501
C06694=1003.608,317.075,-162.020,169.048,54.473,160.500
C06695=1003.603,316.827,-161.989,169.041,54.478,160.500
C06696=1003.599,316.578,-161.957,169.034,54.484,160.500
C06697=1003.594,316.331,-161.927,169.027,54.488,160.499
C06698=1003.589,316.083,-161.896,169.020,54.494,160.499
C06699=1003.584,315.834,-161.865,169.012,54.499,160.498
C06700=1003.579,315.586,-161.834,169.005,54.504,160.498
C06701=1003.575,315.339,-161.803,168.998,54.509,160.497
C06702=1003.570,315.090,-161.772,168.990,54.514,160.497
C06703=1003.565,314.842,-161.741,168.983,54.519,160.496
C06704=1003.560,314.594,-161.710,168.976,54.524,160.496
C06705=1003.556,314.347,-161.679,168.970,54.529,160.495
C06706=1003.551,314.098,-161.648,168.961,54.534,160.495
C06707=1003.546,313.850,-161.617,168.955,54.539,160.494
C06708=1003.542,313.603,-161.586,168.948,54.544,160.494
C06709=1003.537,313.355,-161.555,168.941,54.549,160.494
C06710=1003.532,313.107,-161.525,168.933,54.555,160.493
C06711=1003.528,312.859,-161.493,168.926,54.560,160.493
C06712=1003.523,312.610,-161.463,168.920,54.565,160.492
C06713=1003.519,312.363,-161.432,168.912,54.570,160.492
C06714=1003.514,312.114,-161.401,168.905,54.575,160.491
C06715=1003.509,311.867,-161.371,168.898,54.580,160.491
C06716=1003.505,311.619,-161.339,168.891,54.585,160.491
C06717=1003.501,311.370,-161.309,168.884,54.591,160.490
C06718=1003.495,311.106,-161.277,168.876,54.596,160.490
C06719=1003.491,310.842,-161.244,168.869,54.601,160.489
C06720=1003.486,310.577,-161.211,168.861,54.607,160.489
C06721=1003.481,310.313,-161.179,168.854,54.612,160.488
C06722=1003.234,310.726,-161.596,168.849,54.624,160.490
C06723=1003.241,311.080,-161.638,168.859,54.617,160.490
C06724=1003.247,311.432,-161.682,168.869,54.610,160.491
C06725=1003.254,311.786,-161.727,168.879,54.603,160.492
C06726=1003.260,312.139,-161.770,168.889,54.595,160.492
C06727=1003.265,312.387,-161.800,168.896,54.590,160.493
C06728=1003.269,312.635,-161.832,168.903,54.585,160.493
C06729=1003.274,312.882,-161.862,168.910,54.580,160.494
C06730=1003.278,313.131,-161.892,168.918,54.575,160.494
C06731=1003.284,313.379,-161.923,168.925,54.570,160.495
C06732=1003.288,313.627,-161.954,168.931,54.565,160.495
C06733=1003.292,313.875,-161.986,168.939,54.560,160.496
C06734=1003.297,314.123,-162.016,168.945,54.555,160.496
C06735=1003.302,314.371,-162.047,168.953,54.550,160.497
C06736=1003.307,314.619,-162.078,168.960,54.545,160.497
C06737=1003.311,314.866,-162.109,168.967,54.540,160.497
C06738=1003.316,315.115,-162.140,168.974,54.535,160.498
C06739=1003.321,315.363,-162.171,168.982,54.529,160.498
C06740=1003.325,315.610,-162.202,168.989,54.525,160.499
C06741=1003.330,315.858,-162.233,168.996,54.520,160.499
C06742=1003.336,316.107,-162.264,169.004,54.514,160.500
C06743=1003.340,316.355,-162.295,169.011,54.510,160.500
C06744=1003.344,316.602,-162.326,169.017,54.504,160.501
C06745=1003.349,316.851,-162.357,169.025,54.500,160.501
C06746=1003.355,317.099,-162.388,169.033,54.495,160.502
C06747=1003.360,317.347,-162.418,169.039,54.489,160.502
C06748=1003.364,317.595,-162.450,169.046,54.485,160.503
C06749=1003.368,317.843,-162.481,169.055,54.480,160.503
C06750=1003.374,318.091,-162.512,169.062,54.475,160.504
C06751=1003.076,315.884,-162.601,168.980,54.540,160.500
C06752=1003.072,315.636,-162.569,168.973,54.544,160.500
C06753=1003.067,315.388,-162.538,168.966,54.550,160.499
C06754=1003.062,315.140,-162.508,168.958,54.555,160.499
C06755=1003.057,314.892,-162.477,168.951,54.559,160.498
C06756=1003.053,314.643,-162.446,168.945,54.565,160.498
C06757=1003.049,314.396,-162.415,168.937,54.570,160.497
C06758=1003.044,314.147,-162.384,168.929,54.574,160.497
C06759=1003.039,313.900,-162.354,168.923,54.580,160.497
C06760=1003.034,313.652,-162.323,168.916,54.584,160.496
C06761=1003.029,313.404,-162.292,168.909,54.590,160.496
C06762=1003.026,313.155,-162.261,168.901,54.595,160.495
C06763=1003.021,312.907,-162.230,168.894,54.600,160.495
C06764=1003.016,312.685,-162.203,168.888,54.604,160.494
C06765=1003.013,312.463,-162.176,168.882,54.608,160.494
C06766=1003.008,312.241,-162.148,168.875,54.613,160.493
C06767=1003.004,312.018,-162.120,168.869,54.617,160.493
C06768=1003.000,311.797,-162.093,168.863,54.622,160.493
C06769=1002.996,311.574,-162.066,168.856,54.627,160.492
C06770=1002.992,311.351,-162.039,168.850,54.631,160.492
C06771=1002.988,311.130,-162.011,168.844,54.635,160.491
C06772=1002.742,311.523,-162.425,168.838,54.647,160.493
C06773=1002.747,311.813,-162.461,168.846,54.641,160.493
C06774=1002.752,312.104,-162.497,168.855,54.636,160.494
C06775=1002.758,312.394,-162.532,168.863,54.629,160.494
C06776=1002.762,312.685,-162.569,168.872,54.623,160.495
C06777=1002.767,312.933,-162.600,168.879,54.619,160.495
C06778=1002.771,313.181,-162.630,168.886,54.613,160.496
C06779=1002.777,313.429,-162.660,168.893,54.609,160.496
C06780=1002.781,313.677,-162.691,168.899,54.603,160.497
C06781=952.366,450.117,-214.882,168.899,54.603,160.497
//INST
///DATE 2021/06/17 11:00
///ATTR SC,RW,RJ
////FRAME ROBOT
///GROUP1 RB1
NOP
MOVL C00000 V=800.0 PL=0
MOVL C00001 V=800.0 PL=0
MOVL C00002 V=800.0 PL=0
MOVL C00003 V=800.0 PL=0
MOVL C00004 V=800.0 PL=0
MOVL C00005 V=800.0 PL=0
MOVL C00006 V=800.0 PL=0
MOVL C00007 V=800.0 PL=0
MOVL C00008 V=800.0 PL=0
MOVL C00009 V=800.0 PL=0
MOVL C00010 V=800.0 PL=0
MOVL C00011 V=800.0 PL=0
MOVL C00012 V=800.0 PL=0
MOVL C00013 V=800.0 PL=0
MOVL C00014 V=800.0 PL=0
MOVL C00015 V=800.0 PL=0
MOVL C00016 V=800.0 PL=0
MOVL C00017 V=800.0 PL=0
MOVL C00018 V=800.0 PL=0
MOVL C00019 V=800.0 PL=0
MOVL C00020 V=800.0 PL=0
MOVL C00021 V=800.0 PL=0
MOVL C00022 V=800.0 PL=0
MOVL C00023 V=800.0 PL=0
MOVL C00024 V=800.0 PL=0
MOVL C00025 V=800.0 PL=0
MOVL C00026 V=800.0 PL=0
MOVL C00027 V=800.0 PL=0
MOVL C00028 V=800.0 PL=0
MOVL C00029 V=800.0 PL=0
MOVL C00030 V=800.0 PL=0
MOVL C00031 V=800.0 PL=0
MOVL C00032 V=800.0 PL=0
MOVL C00033 V=800.0 PL=0
MOVL C00034 V=800.0 PL=0
MOVL C00035 V=800.0 PL=0
MOVL C00036 V=800.0 PL=0
MOVL C00037 V=800.0 PL=0
MOVL C00038 V=800.0 PL=0
MOVL C00039 V=800.0 PL=0
MOVL C00040 V=800.0 PL=0
MOVL C00041 V=800.0 PL=0
MOVL C00042 V=800.0 PL=0
MOVL C00043 V=800.0 PL=0
MOVL C00044 V=800.0 PL=0
MOVL C00045 V=800.0 PL=0
MOVL C00046 V=800.0 PL=0
MOVL C00047 V=800.0 PL=0
MOVL C00048 V=800.0 PL=0
MOVL C00049 V=800.0 PL=0
MOVL C00050 V=800.0 PL=0
MOVL C00051 V=800.0 PL=0
MOVL C00052 V=800.0 PL=0
MOVL C00053 V=800.0 PL=0
MOVL C00054 V=800.0 PL=0
MOVL C00055 V=800.0 PL=0
MOVL C00056 V=800.0 PL=0
MOVL C00057 V=800.0 PL=0
MOVL C00058 V=800.0 PL=0
MOVL C00059 V=800.0 PL=0
MOVL C00060 V=800.0 PL=0
MOVL C00061 V=800.0 PL=0
MOVL C00062 V=800.0 PL=0
MOVL C00063 V=800.0 PL=0
MOVL C00064 V=800.0 PL=0
MOVL C00065 V=800.0 PL=0
MOVL C00066 V=800.0 PL=0
MOVL C00067 V=800.0 PL=0
MOVL C00068 V=800.0 PL=0
MOVL C00069 V=800.0 PL=0
MOVL C00070 V=800.0 PL=0
MOVL C00071 V=800.0 PL=0
MOVL C00072 V=800.0 PL=0
MOVL C00073 V=800.0 PL=0
MOVL C00074 V=800.0 PL=0
MOVL C00075 V=800.0 PL=0
MOVL C00076 V=800.0 PL=0
MOVL C00077 V=800.0 PL=0
MOVL C00078 V=800.0 PL=0
MOVL C00079 V=800.0 PL=0
MOVL C00080 V=800.0 PL=0
MOVL C00081 V=800.0 PL=0
MOVL C00082 V=800.0 PL=0
MOVL C00083 V=800.0 PL=0
MOVL C00084 V=800.0 PL=0
MOVL C00085 V=800.0 PL=0
MOVL C00086 V=800.0 PL=0
MOVL C00087 V=800.0 PL=0
MOVL C00088 V=800.0 PL=0
MOVL C00089 V=800.0 PL=0
MOVL C00090 V=800.0 PL=0
MOVL C00091 V=800.0 PL=0
MOVL C00092 V=800.0 PL=0
MOVL C00093 V=800.0 PL=0
MOVL C00094 V=800.0 PL=0
MOVL C00095 V=800.0 PL=0
MOVL C00096 V=800.0 PL=0
MOVL C00097 V=800.0 PL=0
MOVL C00098 V=800.0 PL=0
MOVL C00099 V=800.0 PL=0
MOVL C00100 V=800.0 PL=0
MOVL C00101 V=800.0 PL=0
MOVL C00102 V=800.0 PL=0
MOVL C00103 V=800.0 PL=0
MOVL C00104 V=800.0 PL=0
MOVL C00105 V=800.0 PL=0
MOVL C00106 V=800.0 PL=0
MOVL C00107 V=800.0 PL=0
MOVL C00108 V=800.0 PL=0
MOVL C00109 V=800.0 PL=0
MOVL C00110 V=800.0 PL=0
MOVL C00111 V=800.0 PL=0
MOVL C00112 V=800.0 PL=0
MOVL C00113 V=800.0 PL=0
MOVL C00114 V=800.0 PL=0
MOVL C00115 V=800.0 PL=0
MOVL C00116 V=800.0 PL=0
MOVL C00117 V=800.0 PL=0
MOVL C00118 V=800.0 PL=0
MOVL C00119 V=800.0 PL=0
MOVL C00120 V=800.0 PL=0
MOVL C00121 V=800.0 PL=0
MOVL C00122 V=800.0 PL=0
MOVL C00123 V=800.0 PL=0
MOVL C00124 V=800.0 PL=0
MOVL C00125 V=800.0 PL=0
MOVL C00126 V=800.0 PL=0
MOVL C00127 V=800.0 PL=0
MOVL C00128 V=800.0 PL=0
MOVL C00129 V=800.0 PL=0
MOVL C00130 V=800.0 PL=0
MOVL C00131 V=800.0 PL=0
MOVL C00132 V=800.0 PL=0
MOVL C00133 V=800.0 PL=0
MOVL C00134 V=800.0 PL=0
MOVL C00135 V=800.0 PL=0
MOVL C00136 V=800.0 PL=0
MOVL C00137 V=800.0 PL=0
MOVL C00138 V=800.0 PL=0
MOVL C00139 V=800.0 PL=0
MOVL C00140 V=800.0 PL=0
MOVL C00141 V=800.0 PL=0
MOVL C00142 V=800.0 PL=0
MOVL C00143 V=800.0 PL=0
MOVL C00144 V=800.0 PL=0
MOVL C00145 V=800.0 PL=0
MOVL C00146 V=800.0 PL=0
MOVL C00147 V=800.0 PL=0
MOVL C00148 V=800.0 PL=0
MOVL C00149 V=800.0 PL=0
MOVL C00150 V=800.0 PL=0
MOVL C00151 V=800.0 PL=0
MOVL C00152 V=800.0 PL=0
MOVL C00153 V=800.0 PL=0
MOVL C00154 V=800.0 PL=0
MOVL C00155 V=800.0 PL=0
MOVL C00156 V=800.0 PL=0
MOVL C00157 V=800.0 PL=0
MOVL C00158 V=800.0 PL=0
MOVL C00159 V=800.0 PL=0
MOVL C00160 V=800.0 PL=0
MOVL C00161 V=800.0 PL=0
MOVL C00162 V=800.0 PL=0
MOVL C00163 V=800.0 PL=0
MOVL C00164 V=800.0 PL=0
MOVL C00165 V=800.0 PL=0
MOVL C00166 V=800.0 PL=0
MOVL C00167 V=800.0 PL=0
MOVL C00168 V=800.0 PL=0
MOVL C00169 V=800.0 PL=0
MOVL C00170 V=800.0 PL=0
MOVL C00171 V=800.0 PL=0
MOVL C00172 V=800.0 PL=0
MOVL C00173 V=800.0 PL=0
MOVL C00174 V=800.0 PL=0
MOVL C00175 V=800.0 PL=0
MOVL C00176 V=800.0 PL=0
MOVL C00177 V=800.0 PL=0
MOVL C00178 V=800.0 PL=0
MOVL C00179 V=800.0 PL=0
MOVL C00180 V=800.0 PL=0
MOVL C00181 V=800.0 PL=0
MOVL C00182 V=800.0 PL=0
MOVL C00183 V=800.0 PL=0
MOVL C00184 V=800.0 PL=0
MOVL C00185 V=800.0 PL=0
MOVL C00186 V=800.0 PL=0
MOVL C00187 V=800.0 PL=0
MOVL C00188 V=800.0 PL=0
MOVL C00189 V=800.0 PL=0
MOVL C00190 V=800.0 PL=0
MOVL C00191 V=800.0 PL=0
MOVL C00192 V=800.0 PL=0
MOVL C00193 V=800.0 PL=0
MOVL C00194 V=800.0 PL=0
MOVL C00195 V=800.0 PL=0
MOVL C00196 V=800.0 PL=0
MOVL C00197 V=800.0 PL=0
MOVL C00198 V=800.0 PL=0
MOVL C00199 V=800.0 PL=0
MOVL C00200 V=800.0 PL=0
MOVL C00201 V=800.0 PL=0
MOVL C00202 V=800.0 PL=0
MOVL C00203 V=800.0 PL=0
MOVL C00204 V=800.0 PL=0
MOVL C00205 V=800.0 PL=0
MOVL C00206 V=800.0 PL=0
MOVL C00207 V=800.0 PL=0
MOVL C00208 V=800.0 PL=0
MOVL C00209 V=800.0 PL=0
MOVL C00210 V=800.0 PL=0
MOVL C00211 V=800.0 PL=0
MOVL C00212 V=800.0 PL=0
MOVL C00213 V=800.0 PL=0
MOVL C00214 V=800.0 PL=0
MOVL C00215 V=800.0 PL=0
MOVL C00216 V=800.0 PL=0
MOVL C00217 V=800.0 PL=0
MOVL C00218 V=800.0 PL=0
MOVL C00219 V=800.0 PL=0
MOVL C00220 V=800.0 PL=0
MOVL C00221 V=800.0 PL=0
MOVL C00222 V=800.0 PL=0
MOVL C00223 V=800.0 PL=0
MOVL C00224 V=800.0 PL=0
MOVL C00225 V=800.0 PL=0
MOVL C00226 V=800.0 PL=0
MOVL C00227 V=800.0 PL=0
MOVL C00228 V=800.0 PL=0
MOVL C00229 V=800.0 PL=0
MOVL C00230 V=800.0 PL=0
MOVL C00231 V=800.0 PL=0
MOVL C00232 V=800.0 PL=0
MOVL C00233 V=800.0 PL=0
MOVL C00234 V=800.0 PL=0
MOVL C00235 V=800.0 PL=0
MOVL C00236 V=800.0 PL=0
MOVL C00237 V=800.0 PL=0
MOVL C00238 V=800.0 PL=0
MOVL C00239 V=800.0 PL=0
MOVL C00240 V=800.0 PL=0
MOVL C00241 V=800.0 PL=0
MOVL C00242 V=800.0 PL=0
MOVL C00243 V=800.0 PL=0
MOVL C00244 V=800.0 PL=0
MOVL C00245 V=800.0 PL=0
MOVL C00246 V=800.0 PL=0
MOVL C00247 V=800.0 PL=0
MOVL C00248 V=800.0 PL=0
MOVL C00249 V=800.0 PL=0
MOVL C00250 V=800.0 PL=0
MOVL C00251 V=800.0 PL=0
MOVL C00252 V=800.0 PL=0
MOVL C00253 V=800.0 PL=0
MOVL C00254 V=800.0 PL=0
MOVL C00255 V=800.0 PL=0
MOVL C00256 V=800.0 PL=0
MOVL C00257 V=800.0 PL=0
MOVL C00258 V=800.0 PL=0
MOVL C00259 V=800.0 PL=0
MOVL C00260 V=800.0 PL=0
MOVL C00261 V=800.0 PL=0
MOVL C00262 V=800.0 PL=0
MOVL C00263 V=800.0 PL=0
MOVL C00264 V=800.0 PL=0
MOVL C00265 V=800.0 PL=0
MOVL C00266 V=800.0 PL=0
MOVL C00267 V=800.0 PL=0
MOVL C00268 V=800.0 PL=0
MOVL C00269 V=800.0 PL=0
MOVL C00270 V=800.0 PL=0
MOVL C00271 V=800.0 PL=0
MOVL C00272 V=800.0 PL=0
MOVL C00273 V=800.0 PL=0
MOVL C00274 V=800.0 PL=0
MOVL C00275 V=800.0 PL=0
MOVL C00276 V=800.0 PL=0
MOVL C00277 V=800.0 PL=0
MOVL C00278 V=800.0 PL=0
MOVL C00279 V=800.0 PL=0
MOVL C00280 V=800.0 PL=0
MOVL C00281 V=800.0 PL=0
MOVL C00282 V=800.0 PL=0
MOVL C00283 V=800.0 PL=0
MOVL C00284 V=800.0 PL=0
MOVL C00285 V=800.0 PL=0
MOVL C00286 V=800.0 PL=0
MOVL C00287 V=800.0 PL=0
MOVL C00288 V=800.0 PL=0
MOVL C00289 V=800.0 PL=0
MOVL C00290 V=800.0 PL=0
MOVL C00291 V=800.0 PL=0
MOVL C00292 V=800.0 PL=0
MOVL C00293 V=800.0 PL=0
MOVL C00294 V=800.0 PL=0
MOVL C00295 V=800.0 PL=0
MOVL C00296 V=800.0 PL=0
MOVL C00297 V=800.0 PL=0
MOVL C00298 V=800.0 PL=0
MOVL C00299 V=800.0 PL=0
MOVL C00300 V=800.0 PL=0
MOVL C00301 V=800.0 PL=0
MOVL C00302 V=800.0 PL=0
MOVL C00303 V=800.0 PL=0
MOVL C00304 V=800.0 PL=0
MOVL C00305 V=800.0 PL=0
MOVL C00306 V=800.0 PL=0
MOVL C00307 V=800.0 PL=0
MOVL C00308 V=800.0 PL=0
MOVL C00309 V=800.0 PL=0
MOVL C00310 V=800.0 PL=0
MOVL C00311 V=800.0 PL=0
MOVL C00312 V=800.0 PL=0
MOVL C00313 V=800.0 PL=0
MOVL C00314 V=800.0 PL=0
MOVL C00315 V=800.0 PL=0
MOVL C00316 V=800.0 PL=0
MOVL C00317 V=800.0 PL=0
MOVL C00318 V=800.0 PL=0
MOVL C00319 V=800.0 PL=0
MOVL C00320 V=800.0 PL=0
MOVL C00321 V=800.0 PL=0
MOVL C00322 V=800.0 PL=0
MOVL C00323 V=800.0 PL=0
MOVL C00324 V=800.0 PL=0
MOVL C00325 V=800.0 PL=0
MOVL C00326 V=800.0 PL=0
MOVL C00327 V=800.0 PL=0
MOVL C00328 V=800.0 PL=0
MOVL C00329 V=800.0 PL=0
MOVL C00330 V=800.0 PL=0
MOVL C00331 V=800.0 PL=0
MOVL C00332 V=800.0 PL=0
MOVL C00333 V=800.0 PL=0
MOVL C00334 V=800.0 PL=0
MOVL C00335 V=800.0 PL=0
MOVL C00336 V=800.0 PL=0
MOVL C00337 V=800.0 PL=0
MOVL C00338 V=800.0 PL=0
MOVL C00339 V=800.0 PL=0
MOVL C00340 V=800.0 PL=0
MOVL C00341 V=800.0 PL=0
MOVL C00342 V=800.0 PL=0
MOVL C00343 V=800.0 PL=0
MOVL C00344 V=800.0 PL=0
MOVL C00345 V=800.0 PL=0
MOVL C00346 V=800.0 PL=0
MOVL C00347 V=800.0 PL=0
MOVL C00348 V=800.0 PL=0
MOVL C00349 V=800.0 PL=0
MOVL C00350 V=800.0 PL=0
MOVL C00351 V=800.0 PL=0
MOVL C00352 V=800.0 PL=0
MOVL C00353 V=800.0 PL=0
MOVL C00354 V=800.0 PL=0
MOVL C00355 V=800.0 PL=0
MOVL C00356 V=800.0 PL=0
MOVL C00357 V=800.0 PL=0
MOVL C00358 V=800.0 PL=0
MOVL C00359 V=800.0 PL=0
MOVL C00360 V=800.0 PL=0
MOVL C00361 V=800.0 PL=0
MOVL C00362 V=800.0 PL=0
MOVL C00363 V=800.0 PL=0
MOVL C00364 V=800.0 PL=0
MOVL C00365 V=800.0 PL=0
MOVL C00366 V=800.0 PL=0
MOVL C00367 V=800.0 PL=0
MOVL C00368 V=800.0 PL=0
MOVL C00369 V=800.0 PL=0
MOVL C00370 V=800.0 PL=0
MOVL C00371 V=800.0 PL=0
MOVL C00372 V=800.0 PL=0
MOVL C00373 V=800.0 PL=0
MOVL C00374 V=800.0 PL=0
MOVL C00375 V=800.0 PL=0
MOVL C00376 V=800.0 PL=0
MOVL C00377 V=800.0 PL=0
MOVL C00378 V=800.0 PL=0
MOVL C00379 V=800.0 PL=0
MOVL C00380 V=800.0 PL=0
MOVL C00381 V=800.0 PL=0
MOVL C00382 V=800.0 PL=0
MOVL C00383 V=800.0 PL=0
MOVL C00384 V=800.0 PL=0
MOVL C00385 V=800.0 PL=0
MOVL C00386 V=800.0 PL=0
MOVL C00387 V=800.0 PL=0
MOVL C00388 V=800.0 PL=0
MOVL C00389 V=800.0 PL=0
MOVL C00390 V=800.0 PL=0
MOVL C00391 V=800.0 PL=0
MOVL C00392 V=800.0 PL=0
MOVL C00393 V=800.0 PL=0
MOVL C00394 V=800.0 PL=0
MOVL C00395 V=800.0 PL=0
MOVL C00396 V=800.0 PL=0
MOVL C00397 V=800.0 PL=0
MOVL C00398 V=800.0 PL=0
MOVL C00399 V=800.0 PL=0
MOVL C00400 V=800.0 PL=0
MOVL C00401 V=800.0 PL=0
MOVL C00402 V=800.0 PL=0
MOVL C00403 V=800.0 PL=0
MOVL C00404 V=800.0 PL=0
MOVL C00405 V=800.0 PL=0
MOVL C00406 V=800.0 PL=0
MOVL C00407 V=800.0 PL=0
MOVL C00408 V=800.0 PL=0
MOVL C00409 V=800.0 PL=0
MOVL C00410 V=800.0 PL=0
MOVL C00411 V=800.0 PL=0
MOVL C00412 V=800.0 PL=0
MOVL C00413 V=800.0 PL=0
MOVL C00414 V=800.0 PL=0
MOVL C00415 V=800.0 PL=0
MOVL C00416 V=800.0 PL=0
MOVL C00417 V=800.0 PL=0
MOVL C00418 V=800.0 PL=0
MOVL C00419 V=800.0 PL=0
MOVL C00420 V=800.0 PL=0
MOVL C00421 V=800.0 PL=0
MOVL C00422 V=800.0 PL=0
MOVL C00423 V=800.0 PL=0
MOVL C00424 V=800.0 PL=0
MOVL C00425 V=800.0 PL=0
MOVL C00426 V=800.0 PL=0
MOVL C00427 V=800.0 PL=0
MOVL C00428 V=800.0 PL=0
MOVL C00429 V=800.0 PL=0
MOVL C00430 V=800.0 PL=0
MOVL C00431 V=800.0 PL=0
MOVL C00432 V=800.0 PL=0
MOVL C00433 V=800.0 PL=0
MOVL C00434 V=800.0 PL=0
MOVL C00435 V=800.0 PL=0
MOVL C00436 V=800.0 PL=0
MOVL C00437 V=800.0 PL=0
MOVL C00438 V=800.0 PL=0
MOVL C00439 V=800.0 PL=0
MOVL C00440 V=800.0 PL=0
MOVL C00441 V=800.0 PL=0
MOVL C00442 V=800.0 PL=0
MOVL C00443 V=800.0 PL=0
MOVL C00444 V=800.0 PL=0
MOVL C00445 V=800.0 PL=0
MOVL C00446 V=800.0 PL=0
MOVL C00447 V=800.0 PL=0
MOVL C00448 V=800.0 PL=0
MOVL C00449 V=800.0 PL=0
MOVL C00450 V=800.0 PL=0
MOVL C00451 V=800.0 PL=0
MOVL C00452 V=800.0 PL=0
MOVL C00453 V=800.0 PL=0
MOVL C00454 V=800.0 PL=0
MOVL C00455 V=800.0 PL=0
MOVL C00456 V=800.0 PL=0
MOVL C00457 V=800.0 PL=0
MOVL C00458 V=800.0 PL=0
MOVL C00459 V=800.0 PL=0
MOVL C00460 V=800.0 PL=0
MOVL C00461 V=800.0 PL=0
MOVL C00462 V=800.0 PL=0
MOVL C00463 V=800.0 PL=0
MOVL C00464 V=800.0 PL=0
MOVL C00465 V=800.0 PL=0
MOVL C00466 V=800.0 PL=0
MOVL C00467 V=800.0 PL=0
MOVL C00468 V=800.0 PL=0
MOVL C00469 V=800.0 PL=0
MOVL C00470 V=800.0 PL=0
MOVL C00471 V=800.0 PL=0
MOVL C00472 V=800.0 PL=0
MOVL C00473 V=800.0 PL=0
MOVL C00474 V=800.0 PL=0
MOVL C00475 V=800.0 PL=0
MOVL C00476 V=800.0 PL=0
MOVL C00477 V=800.0 PL=0
MOVL C00478 V=800.0 PL=0
MOVL C00479 V=800.0 PL=0
MOVL C00480 V=800.0 PL=0
MOVL C00481 V=800.0 PL=0
MOVL C00482 V=800.0 PL=0
MOVL C00483 V=800.0 PL=0
MOVL C00484 V=800.0 PL=0
MOVL C00485 V=800.0 PL=0
MOVL C00486 V=800.0 PL=0
MOVL C00487 V=800.0 PL=0
MOVL C00488 V=800.0 PL=0
MOVL C00489 V=800.0 PL=0
MOVL C00490 V=800.0 PL=0
MOVL C00491 V=800.0 PL=0
MOVL C00492 V=800.0 PL=0
MOVL C00493 V=800.0 PL=0
MOVL C00494 V=800.0 PL=0
MOVL C00495 V=800.0 PL=0
MOVL C00496 V=800.0 PL=0
MOVL C00497 V=800.0 PL=0
MOVL C00498 V=800.0 PL=0
MOVL C00499 V=800.0 PL=0
MOVL C00500 V=800.0 PL=0
MOVL C00501 V=800.0 PL=0
MOVL C00502 V=800.0 PL=0
MOVL C00503 V=800.0 PL=0
MOVL C00504 V=800.0 PL=0
MOVL C00505 V=800.0 PL=0
MOVL C00506 V=800.0 PL=0
MOVL C00507 V=800.0 PL=0
MOVL C00508 V=800.0 PL=0
MOVL C00509 V=800.0 PL=0
MOVL C00510 V=800.0 PL=0
MOVL C00511 V=800.0 PL=0
MOVL C00512 V=800.0 PL=0
MOVL C00513 V=800.0 PL=0
MOVL C00514 V=800.0 PL=0
MOVL C00515 V=800.0 PL=0
MOVL C00516 V=800.0 PL=0
MOVL C00517 V=800.0 PL=0
MOVL C00518 V=800.0 PL=0
MOVL C00519 V=800.0 PL=0
MOVL C00520 V=800.0 PL=0
MOVL C00521 V=800.0 PL=0
MOVL C00522 V=800.0 PL=0
MOVL C00523 V=800.0 PL=0
MOVL C00524 V=800.0 PL=0
MOVL C00525 V=800.0 PL=0
MOVL C00526 V=800.0 PL=0
MOVL C00527 V=800.0 PL=0
MOVL C00528 V=800.0 PL=0
MOVL C00529 V=800.0 PL=0
MOVL C00530 V=800.0 PL=0
MOVL C00531 V=800.0 PL=0
MOVL C00532 V=800.0 PL=0
MOVL C00533 V=800.0 PL=0
MOVL C00534 V=800.0 PL=0
MOVL C00535 V=800.0 PL=0
MOVL C00536 V=800.0 PL=0
MOVL C00537 V=800.0 PL=0
MOVL C00538 V=800.0 PL=0
MOVL C00539 V=800.0 PL=0
MOVL C00540 V=800.0 PL=0
MOVL C00541 V=800.0 PL=0
MOVL C00542 V=800.0 PL=0
MOVL C00543 V=800.0 PL=0
MOVL C00544 V=800.0 PL=0
MOVL C00545 V=800.0 PL=0
MOVL C00546 V=800.0 PL=0
MOVL C00547 V=800.0 PL=0
MOVL C00548 V=800.0 PL=0
MOVL C00549 V=800.0 PL=0
MOVL C00550 V=800.0 PL=0
MOVL C00551 V=800.0 PL=0
MOVL C00552 V=800.0 PL=0
MOVL C00553 V=800.0 PL=0
MOVL C00554 V=800.0 PL=0
MOVL C00555 V=800.0 PL=0
MOVL C00556 V=800.0 PL=0
MOVL C00557 V=800.0 PL=0
MOVL C00558 V=800.0 PL=0
MOVL C00559 V=800.0 PL=0
MOVL C00560 V=800.0 PL=0
MOVL C00561 V=800.0 PL=0
MOVL C00562 V=800.0 PL=0
MOVL C00563 V=800.0 PL=0
MOVL C00564 V=800.0 PL=0
MOVL C00565 V=800.0 PL=0
MOVL C00566 V=800.0 PL=0
MOVL C00567 V=800.0 PL=0
MOVL C00568 V=800.0 PL=0
MOVL C00569 V=800.0 PL=0
MOVL C00570 V=800.0 PL=0
MOVL C00571 V=800.0 PL=0
MOVL C00572 V=800.0 PL=0
MOVL C00573 V=800.0 PL=0
MOVL C00574 V=800.0 PL=0
MOVL C00575 V=800.0 PL=0
MOVL C00576 V=800.0 PL=0
MOVL C00577 V=800.0 PL=0
MOVL C00578 V=800.0 PL=0
MOVL C00579 V=800.0 PL=0
MOVL C00580 V=800.0 PL=0
MOVL C00581 V=800.0 PL=0
MOVL C00582 V=800.0 PL=0
MOVL C00583 V=800.0 PL=0
MOVL C00584 V=800.0 PL=0
MOVL C00585 V=800.0 PL=0
MOVL C00586 V=800.0 PL=0
MOVL C00587 V=800.0 PL=0
MOVL C00588 V=800.0 PL=0
MOVL C00589 V=800.0 PL=0
MOVL C00590 V=800.0 PL=0
MOVL C00591 V=800.0 PL=0
MOVL C00592 V=800.0 PL=0
MOVL C00593 V=800.0 PL=0
MOVL C00594 V=800.0 PL=0
MOVL C00595 V=800.0 PL=0
MOVL C00596 V=800.0 PL=0
MOVL C00597 V=800.0 PL=0
MOVL C00598 V=800.0 PL=0
MOVL C00599 V=800.0 PL=0
MOVL C00600 V=800.0 PL=0
MOVL C00601 V=800.0 PL=0
MOVL C00602 V=800.0 PL=0
MOVL C00603 V=800.0 PL=0
MOVL C00604 V=800.0 PL=0
MOVL C00605 V=800.0 PL=0
MOVL C00606 V=800.0 PL=0
MOVL C00607 V=800.0 PL=0
MOVL C00608 V=800.0 PL=0
MOVL C00609 V=800.0 PL=0
MOVL C00610 V=800.0 PL=0
MOVL C00611 V=800.0 PL=0
MOVL C00612 V=800.0 PL=0
MOVL C00613 V=800.0 PL=0
MOVL C00614 V=800.0 PL=0
MOVL C00615 V=800.0 PL=0
MOVL C00616 V=800.0 PL=0
MOVL C00617 V=800.0 PL=0
MOVL C00618 V=800.0 PL=0
MOVL C00619 V=800.0 PL=0
MOVL C00620 V=800.0 PL=0
MOVL C00621 V=800.0 PL=0
MOVL C00622 V=800.0 PL=0
MOVL C00623 V=800.0 PL=0
MOVL C00624 V=800.0 PL=0
MOVL C00625 V=800.0 PL=0
MOVL C00626 V=800.0 PL=0
MOVL C00627 V=800.0 PL=0
MOVL C00628 V=800.0 PL=0
MOVL C00629 V=800.0 PL=0
MOVL C00630 V=800.0 PL=0
MOVL C00631 V=800.0 PL=0
MOVL C00632 V=800.0 PL=0
MOVL C00633 V=800.0 PL=0
MOVL C00634 V=800.0 PL=0
MOVL C00635 V=800.0 PL=0
MOVL C00636 V=800.0 PL=0
MOVL C00637 V=800.0 PL=0
MOVL C00638 V=800.0 PL=0
MOVL C00639 V=800.0 PL=0
MOVL C00640 V=800.0 PL=0
MOVL C00641 V=800.0 PL=0
MOVL C00642 V=800.0 PL=0
MOVL C00643 V=800.0 PL=0
MOVL C00644 V=800.0 PL=0
MOVL C00645 V=800.0 PL=0
MOVL C00646 V=800.0 PL=0
MOVL C00647 V=800.0 PL=0
MOVL C00648 V=800.0 PL=0
MOVL C00649 V=800.0 PL=0
MOVL C00650 V=800.0 PL=0
MOVL C00651 V=800.0 PL=0
MOVL C00652 V=800.0 PL=0
MOVL C00653 V=800.0 PL=0
MOVL C00654 V=800.0 PL=0
MOVL C00655 V=800.0 PL=0
MOVL C00656 V=800.0 PL=0
MOVL C00657 V=800.0 PL=0
MOVL C00658 V=800.0 PL=0
MOVL C00659 V=800.0 PL=0
MOVL C00660 V=800.0 PL=0
MOVL C00661 V=800.0 PL=0
MOVL C00662 V=800.0 PL=0
MOVL C00663 V=800.0 PL=0
MOVL C00664 V=800.0 PL=0
MOVL C00665 V=800.0 PL=0
MOVL C00666 V=800.0 PL=0
MOVL C00667 V=800.0 PL=0
MOVL C00668 V=800.0 PL=0
MOVL C00669 V=800.0 PL=0
MOVL C00670 V=800.0 PL=0
MOVL C00671 V=800.0 PL=0
MOVL C00672 V=800.0 PL=0
MOVL C00673 V=800.0 PL=0
MOVL C00674 V=800.0 PL=0
MOVL C00675 V=800.0 PL=0
MOVL C00676 V=800.0 PL=0
MOVL C00677 V=800.0 PL=0
MOVL C00678 V=800.0 PL=0
MOVL C00679 V=800.0 PL=0
MOVL C00680 V=800.0 PL=0
MOVL C00681 V=800.0 PL=0
MOVL C00682 V=800.0 PL=0
MOVL C00683 V=800.0 PL=0
MOVL C00684 V=800.0 PL=0
MOVL C00685 V=800.0 PL=0
MOVL C00686 V=800.0 PL=0
MOVL C00687 V=800.0 PL=0
MOVL C00688 V=800.0 PL=0
MOVL C00689 V=800.0 PL=0
MOVL C00690 V=800.0 PL=0
MOVL C00691 V=800.0 PL=0
MOVL C00692 V=800.0 PL=0
MOVL C00693 V=800.0 PL=0
MOVL C00694 V=800.0 PL=0
MOVL C00695 V=800.0 PL=0
MOVL C00696 V=800.0 PL=0
MOVL C00697 V=800.0 PL=0
MOVL C00698 V=800.0 PL=0
MOVL C00699 V=800.0 PL=0
MOVL C00700 V=800.0 PL=0
MOVL C00701 V=800.0 PL=0
MOVL C00702 V=800.0 PL=0
MOVL C00703 V=800.0 PL=0
MOVL C00704 V=800.0 PL=0
MOVL C00705 V=800.0 PL=0
MOVL C00706 V=800.0 PL=0
MOVL C00707 V=800.0 PL=0
MOVL C00708 V=800.0 PL=0
MOVL C00709 V=800.0 PL=0
MOVL C00710 V=800.0 PL=0
MOVL C00711 V=800.0 PL=0
MOVL C00712 V=800.0 PL=0
MOVL C00713 V=800.0 PL=0
MOVL C00714 V=800.0 PL=0
MOVL C00715 V=800.0 PL=0
MOVL C00716 V=800.0 PL=0
MOVL C00717 V=800.0 PL=0
MOVL C00718 V=800.0 PL=0
MOVL C00719 V=800.0 PL=0
MOVL C00720 V=800.0 PL=0
MOVL C00721 V=800.0 PL=0
MOVL C00722 V=800.0 PL=0
MOVL C00723 V=800.0 PL=0
MOVL C00724 V=800.0 PL=0
MOVL C00725 V=800.0 PL=0
MOVL C00726 V=800.0 PL=0
MOVL C00727 V=800.0 PL=0
MOVL C00728 V=800.0 PL=0
MOVL C00729 V=800.0 PL=0
MOVL C00730 V=800.0 PL=0
MOVL C00731 V=800.0 PL=0
MOVL C00732 V=800.0 PL=0
MOVL C00733 V=800.0 PL=0
MOVL C00734 V=800.0 PL=0
MOVL C00735 V=800.0 PL=0
MOVL C00736 V=800.0 PL=0
MOVL C00737 V=800.0 PL=0
MOVL C00738 V=800.0 PL=0
MOVL C00739 V=800.0 PL=0
MOVL C00740 V=800.0 PL=0
MOVL C00741 V=800.0 PL=0
MOVL C00742 V=800.0 PL=0
MOVL C00743 V=800.0 PL=0
MOVL C00744 V=800.0 PL=0
MOVL C00745 V=800.0 PL=0
MOVL C00746 V=800.0 PL=0
MOVL C00747 V=800.0 PL=0
MOVL C00748 V=800.0 PL=0
MOVL C00749 V=800.0 PL=0
MOVL C00750 V=800.0 PL=0
MOVL C00751 V=800.0 PL=0
MOVL C00752 V=800.0 PL=0
MOVL C00753 V=800.0 PL=0
MOVL C00754 V=800.0 PL=0
MOVL C00755 V=800.0 PL=0
MOVL C00756 V=800.0 PL=0
MOVL C00757 V=800.0 PL=0
MOVL C00758 V=800.0 PL=0
MOVL C00759 V=800.0 PL=0
MOVL C00760 V=800.0 PL=0
MOVL C00761 V=800.0 PL=0
MOVL C00762 V=800.0 PL=0
MOVL C00763 V=800.0 PL=0
MOVL C00764 V=800.0 PL=0
MOVL C00765 V=800.0 PL=0
MOVL C00766 V=800.0 PL=0
MOVL C00767 V=800.0 PL=0
MOVL C00768 V=800.0 PL=0
MOVL C00769 V=800.0 PL=0
MOVL C00770 V=800.0 PL=0
MOVL C00771 V=800.0 PL=0
MOVL C00772 V=800.0 PL=0
MOVL C00773 V=800.0 PL=0
MOVL C00774 V=800.0 PL=0
MOVL C00775 V=800.0 PL=0
MOVL C00776 V=800.0 PL=0
MOVL C00777 V=800.0 PL=0
MOVL C00778 V=800.0 PL=0
MOVL C00779 V=800.0 PL=0
MOVL C00780 V=800.0 PL=0
MOVL C00781 V=800.0 PL=0
MOVL C00782 V=800.0 PL=0
MOVL C00783 V=800.0 PL=0
